KUKA KRL program: EPS_2_25694_WD01A_A_20260120031656.src

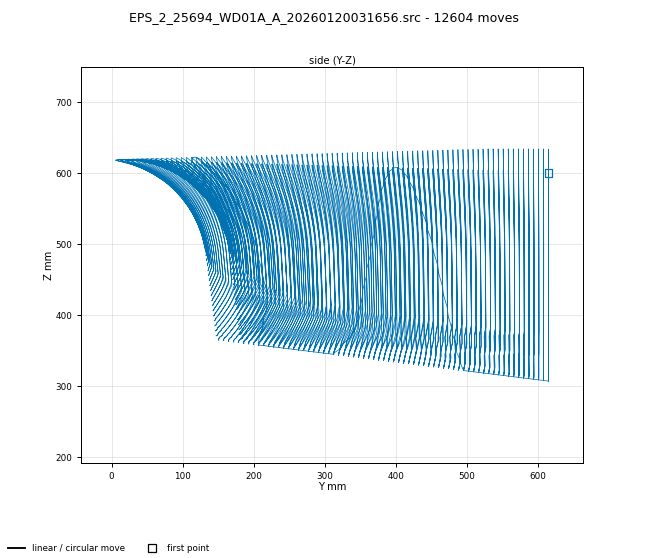
[picture p0: tool path of EPS_2_25694_WD01A_A_20260120031656.src, 12604 of 12606 moves have a stored position in this frame; points joined in program order, loops and branches not executed]
&ACCESS RVP
&REL 4
&COMMENT QRS 19112012
&PARAM EDITMASK = *
DEF PART()
EXT BAS (BAS_COMMAND :IN,REAL :IN )
INT I
BAS (#INITMOV,0 )

;KUKA QRS Post kuka4.cps  Date:22-06-2017 !

File_ID=2994

QRS_PRE_INIT()

;Init var - Until changes are made in qrs_pre_init
Outlet_Square_prg=0
Inlet_1_Square_prg=0
Inlet_2_Square_prg=0
Inlet_3_Square_prg=0
Inlet_4_Square_prg=0
Inlet_5_Square_prg=0

Outlet_1={X 0.000, Y 527.380, Z 509.000, B 0.000, E1 0.000 }
Inlet_1={X 0.000, Y 529.540, Z 479.000, B 0.000, E1 175.000 }
Outlet_1_type=251
Inlet_1_type=251
;QRS#1=Sidecore dimensions
;QRS#2=250-10" PVC SDR 35
;QRS#3=250-10" PVC SDR 35
;QRS#4=
;QRS#5=
;QRS#6=
;QRS#7=
;QRS#8=
;QRS#9=14M PSX
;QRS#10=14M PSX
;QRS#11=
;QRS#12=
;QRS#13=
;QRS#14=
;QRS#15=
;QRS#16=1220x127x914 3'
;QRS#17=EPS Height
;QRS#18=634,5
;QRS#19=*
;QRS#20= UPDATED VERSION 22-06-2017
;QRS#21=*
Outlet_Square=0100
Inlet_1_Square=0100
Inlet_2_Square=0
Inlet_3_Square=0
Inlet_4_Square=0
Inlet_5_Square=0
Mill_Square=1
Outlet_Square_Prg=205
Inlet_1_Square_prg=205

QRS_INIT()

$ADVANCE=5

; T1
PTP {E1 173.652,E2 173.652}
PTP {X 0,Y 615.445,A -85,B 0,C 180,E1 173.652,E2 173.652,E3 0,E4 0,E5 0,E6 0}
QRS_SPEED_INIT()
LIN {X 0,Y 615.445,Z 600,A -85,B 0,C 180,E1 173.652,E2 173.652,E3 0,E4 0,E5 0,E6 0} C_VEL
LIN {X 0,Y 615.445,Z 317.5,A -85,B 0,C 180,E1 173.652,E2 173.652} C_VEL
LIN {X 0,Y 615.445,Z 309.32,A -85,B 0,C 180,E1 173.652,E2 173.652} C_VEL
LIN {X 0,Y 615.438,Z 307.32,A -85,B 0,C 180,E1 173.466,E2 173.466} C_VEL
LIN {X 0,Y 615.464,Z 307.316,A -85,B 0,C 180,E1 170.801,E2 170.801} C_VEL
LIN {X 0,Y 615.478,Z 307.325,A -85,B 0,C 180,E1 168.139,E2 168.139} C_VEL
LIN {X 0,Y 615.433,Z 307.32,A -85,B 0,C 180,E1 165.449,E2 165.449} C_VEL
LIN {X 0,Y 615.481,Z 307.316,A -85,B 0,C 180,E1 162.729,E2 162.729} C_VEL
LIN {X 0,Y 615.451,Z 307.323,A -85,B 0,C 180,E1 159.966,E2 159.966} C_VEL
LIN {X 0,Y 615.43,Z 307.322,A -85,B 0,C 180,E1 157.668,E2 157.668} C_VEL
LIN {X 0,Y 615.429,Z 307.322,A -85,B 0,C 180,E1 155.725,E2 155.725} C_VEL
LIN {X 0,Y 615.426,Z 307.322,A -85,B 0,C 180,E1 153.553,E2 153.553} C_VEL
LIN {X 0,Y 615.493,Z 307.323,A -85,B 0,C 180,E1 150.594,E2 150.594} C_VEL
LIN {X 0,Y 615.471,Z 307.324,A -85,B 0,C 180,E1 148.313,E2 148.313} C_VEL
LIN {X 0,Y 615.433,Z 307.323,A -85,B 0,C 180,E1 145.974,E2 145.974} C_VEL
LIN {X 0,Y 615.421,Z 307.322,A -85,B 0,C 180,E1 143.57,E2 143.57} C_VEL
LIN {X 0,Y 615.463,Z 307.322,A -85,B 0,C 180,E1 140.941,E2 140.941} C_VEL
LIN {X 0,Y 615.482,Z 307.325,A -85,B 0,C 180,E1 138.525,E2 138.525} C_VEL
LIN {X 0,Y 615.424,Z 307.324,A -85,B 0,C 180,E1 136.009,E2 136.009} C_VEL
LIN {X 0,Y 615.421,Z 307.324,A -85,B 0,C 180,E1 133.99,E2 133.99} C_VEL
LIN {X 0,Y 615.419,Z 307.324,A -85,B 0,C 180,E1 131.48,E2 131.48} C_VEL
LIN {X 0,Y 615.473,Z 307.326,A -85,B 0,C 180,E1 128.906,E2 128.906} C_VEL
LIN {X 0,Y 615.446,Z 307.325,A -85,B 0,C 180,E1 126.428,E2 126.428} C_VEL
LIN {X 0,Y 615.414,Z 307.325,A -85,B 0,C 180,E1 124.027,E2 124.027} C_VEL
LIN {X 0,Y 615.412,Z 307.325,A -85,B 0,C 180,E1 121.69,E2 121.69} C_VEL
LIN {X 0,Y 615.428,Z 307.325,A -85,B 0,C 180,E1 119.41,E2 119.41} C_VEL
LIN {X 0,Y 615.444,Z 307.323,A -85,B 0,C 180,E1 116.446,E2 116.446} C_VEL
LIN {X 0,Y 615.423,Z 307.397,A -85,B 0,C 180,E1 115.597,E2 115.597} C_VEL
LIN {X 0,Y 615.49,Z 326.441,A -85,B 0,C 180,E1 112.845,E2 112.845} C_VEL
LIN {X 0,Y 615.48,Z 342.634,A -85,B 0,C 180,E1 110.538,E2 110.538} C_VEL
LIN {X 0,Y 615.496,Z 479.164,A -85,B 0,C 180,E1 108.905,E2 108.905} C_VEL
LIN {X 0,Y 615.495,Z 493.339,A -85,B 0,C 180,E1 108.605,E2 108.605} C_VEL
LIN {X 0,Y 615.494,Z 506.524,A -85,B 0,C 180,E1 108.2,E2 108.2} C_VEL
LIN {X 0,Y 615.497,Z 518.867,A -85,B 0,C 180,E1 107.699,E2 107.699} C_VEL
LIN {X 0,Y 615.492,Z 532.079,A -85,B 0,C 180,E1 107.014,E2 107.014} C_VEL
LIN {X 0,Y 615.498,Z 543.22,A -85,B 0,C 180,E1 106.301,E2 106.301} C_VEL
LIN {X 0,Y 615.499,Z 554.818,A -85,B 0,C 180,E1 105.395,E2 105.395} C_VEL
LIN {X 0,Y 615.496,Z 565.347,A -85,B 0,C 180,E1 104.395,E2 104.395} C_VEL
LIN {X 0,Y 615.497,Z 574.255,A -85,B 0,C 180,E1 103.369,E2 103.369} C_VEL
LIN {X 0,Y 615.496,Z 582.577,A -85,B 0,C 180,E1 102.195,E2 102.195} C_VEL
LIN {X 0,Y 615.496,Z 588.372,A -85,B 0,C 180,E1 101.193,E2 101.193} C_VEL
LIN {X 0,Y 615.497,Z 593.088,A -85,B 0,C 180,E1 100.194,E2 100.194} C_VEL
LIN {X 0,Y 615.497,Z 597.952,A -85,B 0,C 180,E1 98.868,E2 98.868} C_VEL
LIN {X 0,Y 615.496,Z 600.595,A -85,B 0,C 180,E1 97.876,E2 97.876} C_VEL
LIN {X 0,Y 615.495,Z 602.88,A -85,B 0,C 180,E1 96.557,E2 96.557} C_VEL
LIN {X 0,Y 615.489,Z 603.827,A -85,B 0,C 180,E1 95.241,E2 95.241} C_VEL
LIN {X 0,Y 615.493,Z 603.459,A -85,B 0,C 180,E1 93.929,E2 93.929} C_VEL
LIN {X 0,Y 615.491,Z 601.783,A -85,B 0,C 180,E1 92.618,E2 92.618} C_VEL
LIN {X 0,Y 615.495,Z 598.753,A -85,B 0,C 180,E1 91.309,E2 91.309} C_VEL
LIN {X 0,Y 615.496,Z 594.297,A -85,B 0,C 180,E1 90,E2 90} C_VEL
LIN {X 0,Y 615.495,Z 589.885,A -85,B 0,C 180,E1 89.019,E2 89.019} C_VEL
LIN {X 0,Y 615.499,Z 584.538,A -85,B 0,C 180,E1 88.037,E2 88.037} C_VEL
LIN {X 0,Y 615.496,Z 576.898,A -85,B 0,C 180,E1 86.891,E2 86.891} C_VEL
LIN {X 0,Y 615.496,Z 567.474,A -85,B 0,C 180,E1 85.744,E2 85.744} C_VEL
LIN {X 0,Y 615.498,Z 557.621,A -85,B 0,C 180,E1 84.759,E2 84.759} C_VEL
LIN {X 0,Y 615.499,Z 546.628,A -85,B 0,C 180,E1 83.855,E2 83.855} C_VEL
LIN {X 0,Y 615.491,Z 534.195,A -85,B 0,C 180,E1 83.022,E2 83.022} C_VEL
LIN {X 0,Y 615.494,Z 522.224,A -85,B 0,C 180,E1 82.372,E2 82.372} C_VEL
LIN {X 0,Y 615.493,Z 508.759,A -85,B 0,C 180,E1 81.794,E2 81.794} C_VEL
LIN {X 0,Y 615.495,Z 494.585,A -85,B 0,C 180,E1 81.339,E2 81.339} C_VEL
LIN {X 0,Y 615.495,Z 480.493,A -85,B 0,C 180,E1 81.029,E2 81.029} C_VEL
LIN {X 0,Y 615.476,Z 440.355,A -85,B 0,C 180,E1 80.532,E2 80.532} C_VEL
LIN {X 0,Y 615.486,Z 342.551,A -85,B 0,C 180,E1 79.361,E2 79.361} C_VEL
LIN {X 0,Y 615.487,Z 323.409,A -85,B 0,C 180,E1 76.631,E2 76.631} C_VEL
LIN {X 0,Y 615.424,Z 307.324,A -85,B 0,C 180,E1 74.284,E2 74.284} C_VEL
LIN {X 0,Y 615.414,Z 307.324,A -85,B 0,C 180,E1 72.041,E2 72.041} C_VEL
LIN {X 0,Y 615.476,Z 307.322,A -85,B 0,C 180,E1 69.269,E2 69.269} C_VEL
LIN {X 0,Y 615.424,Z 307.324,A -85,B 0,C 180,E1 66.441,E2 66.441} C_VEL
LIN {X 0,Y 615.414,Z 307.325,A -85,B 0,C 180,E1 64.281,E2 64.281} C_VEL
LIN {X 0,Y 615.409,Z 307.325,A -85,B 0,C 180,E1 62.081,E2 62.081} C_VEL
LIN {X 0,Y 615.485,Z 307.325,A -85,B 0,C 180,E1 59.08,E2 59.08} C_VEL
LIN {X 0,Y 615.416,Z 307.325,A -85,B 0,C 180,E1 56.477,E2 56.477} C_VEL
LIN {X 0,Y 615.413,Z 307.325,A -85,B 0,C 180,E1 54.379,E2 54.379} C_VEL
LIN {X 0,Y 615.422,Z 307.324,A -85,B 0,C 180,E1 51.926,E2 51.926} C_VEL
LIN {X 0,Y 615.469,Z 307.328,A -85,B 0,C 180,E1 49.392,E2 49.392} C_VEL
LIN {X 0,Y 615.436,Z 307.323,A -85,B 0,C 180,E1 46.751,E2 46.751} C_VEL
LIN {X 0,Y 615.418,Z 307.324,A -85,B 0,C 180,E1 44.156,E2 44.156} C_VEL
LIN {X 0,Y 615.425,Z 307.323,A -85,B 0,C 180,E1 42.073,E2 42.073} C_VEL
LIN {X 0,Y 615.453,Z 307.324,A -85,B 0,C 180,E1 39.753,E2 39.753} C_VEL
LIN {X 0,Y 615.451,Z 307.32,A -85,B 0,C 180,E1 36.932,E2 36.932} C_VEL
LIN {X 0,Y 615.432,Z 307.321,A -85,B 0,C 180,E1 34.693,E2 34.693} C_VEL
LIN {X 0,Y 615.426,Z 307.322,A -85,B 0,C 180,E1 32.321,E2 32.321} C_VEL
LIN {X 0,Y 615.464,Z 307.324,A -85,B 0,C 180,E1 29.79,E2 29.79} C_VEL
LIN {X 0,Y 615.459,Z 307.318,A -85,B 0,C 180,E1 27.039,E2 27.039} C_VEL
LIN {X 0,Y 615.449,Z 307.319,A -85,B 0,C 180,E1 24.994,E2 24.994} C_VEL
LIN {X 0,Y 615.437,Z 307.32,A -85,B 0,C 180,E1 22.847,E2 22.847} C_VEL
LIN {X 0,Y 615.431,Z 307.32,A -85,B 0,C 180,E1 20.542,E2 20.542} C_VEL
LIN {X 0,Y 615.464,Z 307.323,A -85,B 0,C 180,E1 17.958,E2 17.958} C_VEL
LIN {X 0,Y 615.474,Z 307.316,A -85,B 0,C 180,E1 15.227,E2 15.227} C_VEL
LIN {X 0,Y 615.436,Z 307.32,A -85,B 0,C 180,E1 12.531,E2 12.531} C_VEL
LIN {X 0,Y 615.489,Z 307.325,A -85,B 0,C 180,E1 9.862,E2 9.862} C_VEL
LIN {X 0,Y 615.469,Z 307.315,A -85,B 0,C 180,E1 7.216,E2 7.216} C_VEL
LIN {X 0,Y 615.44,Z 307.319,A -85,B 0,C 180,E1 4.585,E2 4.585} C_VEL
LIN {X 0,Y 615.489,Z 307.324,A -85,B 0,C 180,E1 1.963,E2 1.963} C_VEL
LIN {X 0,Y 615.477,Z 307.314,A -85,B 0,C 180,E1 -0.654,E2 -0.654} C_VEL
LIN {X 0,Y 615.441,Z 307.319,A -85,B 0,C 180,E1 -3.273,E2 -3.273} C_VEL
LIN {X 0,Y 615.483,Z 307.324,A -85,B 0,C 180,E1 -5.898,E2 -5.898} C_VEL
LIN {X 0,Y 615.482,Z 307.313,A -85,B 0,C 180,E1 -8.537,E2 -8.537} C_VEL
LIN {X 0,Y 615.447,Z 307.318,A -85,B 0,C 180,E1 -11.194,E2 -11.194} C_VEL
LIN {X 0,Y 615.498,Z 307.325,A -85,B 0,C 180,E1 -13.935,E2 -13.935} C_VEL
LIN {X 0,Y 615.476,Z 307.312,A -85,B 0,C 180,E1 -16.587,E2 -16.587} C_VEL
LIN {X 0,Y 615.472,Z 307.312,A -85,B 0,C 180,E1 -18.646,E2 -18.646} C_VEL
LIN {X 0,Y 615.465,Z 307.313,A -85,B 0,C 180,E1 -20.731,E2 -20.731} C_VEL
LIN {X 0,Y 615.458,Z 307.314,A -85,B 0,C 180,E1 -22.846,E2 -22.846} C_VEL
LIN {X 0,Y 615.477,Z 307.323,A -85,B 0,C 180,E1 -25.566,E2 -25.566} C_VEL
LIN {X 0,Y 615.488,Z 307.309,A -85,B 0,C 180,E1 -28.45,E2 -28.45} C_VEL
LIN {X 0,Y 615.457,Z 307.317,A -85,B 0,C 180,E1 -31.081,E2 -31.081} C_VEL
LIN {X 0,Y 615.479,Z 307.324,A -85,B 0,C 180,E1 -33.532,E2 -33.532} C_VEL
LIN {X 0,Y 615.484,Z 307.309,A -85,B 0,C 180,E1 -36.425,E2 -36.425} C_VEL
LIN {X 0,Y 615.461,Z 307.317,A -85,B 0,C 180,E1 -39.059,E2 -39.059} C_VEL
LIN {X 0,Y 615.486,Z 307.324,A -85,B 0,C 180,E1 -41.474,E2 -41.474} C_VEL
LIN {X 0,Y 615.494,Z 307.309,A -85,B 0,C 180,E1 -44.149,E2 -44.149} C_VEL
LIN {X 0,Y 615.463,Z 307.317,A -85,B 0,C 180,E1 -46.955,E2 -46.955} C_VEL
LIN {X 0,Y 615.491,Z 307.324,A -85,B 0,C 180,E1 -49.394,E2 -49.394} C_VEL
LIN {X 0,Y 615.488,Z 307.312,A -85,B 0,C 180,E1 -51.988,E2 -51.988} C_VEL
LIN {X 0,Y 615.483,Z 307.308,A -85,B 0,C 180,E1 -54.384,E2 -54.384} C_VEL
LIN {X 0,Y 615.467,Z 307.315,A -85,B 0,C 180,E1 -56.762,E2 -56.762} C_VEL
LIN {X 0,Y 615.476,Z 307.321,A -85,B 0,C 180,E1 -59.079,E2 -59.079} C_VEL
LIN {X 0,Y 615.487,Z 307.32,A -85,B 0,C 180,E1 -61.55,E2 -61.55} C_VEL
LIN {X 0,Y 615.477,Z 307.31,A -85,B 0,C 180,E1 -64.433,E2 -64.433} C_VEL
LIN {X 0,Y 615.474,Z 307.366,A -85,B 0,C 180,E1 -66.51,E2 -66.51} C_VEL
LIN {X 0,Y 615.496,Z 329.445,A -85,B 0,C 180,E1 -69.269,E2 -69.269} C_VEL
LIN {X 0,Y 615.498,Z 352.034,A -85,B 0,C 180,E1 -72.043,E2 -72.043} C_VEL
LIN {X 0,Y 615.49,Z 371.425,A -85,B 0,C 180,E1 -74.392,E2 -74.392} C_VEL
LIN {X 0,Y 615.498,Z 509.933,A -85,B 0,C 180,E1 -76.064,E2 -76.064} C_VEL
LIN {X 0,Y 615.495,Z 524.374,A -85,B 0,C 180,E1 -76.378,E2 -76.378} C_VEL
LIN {X 0,Y 615.489,Z 537.686,A -85,B 0,C 180,E1 -76.799,E2 -76.799} C_VEL
LIN {X 0,Y 615.498,Z 551.58,A -85,B 0,C 180,E1 -77.386,E2 -77.386} C_VEL
LIN {X 0,Y 615.495,Z 564.006,A -85,B 0,C 180,E1 -78.056,E2 -78.056} C_VEL
LIN {X 0,Y 615.499,Z 575.339,A -85,B 0,C 180,E1 -78.807,E2 -78.807} C_VEL
LIN {X 0,Y 615.498,Z 585.747,A -85,B 0,C 180,E1 -79.64,E2 -79.64} C_VEL
LIN {X 0,Y 615.496,Z 596.088,A -85,B 0,C 180,E1 -80.636,E2 -80.636} C_VEL
LIN {X 0,Y 615.497,Z 604.602,A -85,B 0,C 180,E1 -81.629,E2 -81.629} C_VEL
LIN {X 0,Y 615.496,Z 612.726,A -85,B 0,C 180,E1 -82.784,E2 -82.784} C_VEL
LIN {X 0,Y 615.496,Z 618.43,A -85,B 0,C 180,E1 -83.773,E2 -83.773} C_VEL
LIN {X 0,Y 615.495,Z 623.08,A -85,B 0,C 180,E1 -84.759,E2 -84.759} C_VEL
LIN {X 0,Y 615.494,Z 627.901,A -85,B 0,C 180,E1 -86.072,E2 -86.072} C_VEL
LIN {X 0,Y 615.496,Z 631.252,A -85,B 0,C 180,E1 -87.382,E2 -87.382} C_VEL
LIN {X 0,Y 615.489,Z 633.229,A -85,B 0,C 180,E1 -88.691,E2 -88.691} C_VEL
LIN {X 0,Y 615.493,Z 633.889,A -85,B 0,C 180,E1 -90,E2 -90} C_VEL
LIN {X 0,Y 615.489,Z 633.229,A -85,B 0,C 180,E1 -91.309,E2 -91.309} C_VEL
LIN {X 0,Y 615.496,Z 631.252,A -85,B 0,C 180,E1 -92.618,E2 -92.618} C_VEL
LIN {X 0,Y 615.494,Z 627.901,A -85,B 0,C 180,E1 -93.929,E2 -93.929} C_VEL
LIN {X 0,Y 615.495,Z 623.08,A -85,B 0,C 180,E1 -95.241,E2 -95.241} C_VEL
LIN {X 0,Y 615.496,Z 616.628,A -85,B 0,C 180,E1 -96.557,E2 -96.557} C_VEL
LIN {X 0,Y 615.497,Z 609.44,A -85,B 0,C 180,E1 -97.711,E2 -97.711} C_VEL
LIN {X 0,Y 615.497,Z 601.902,A -85,B 0,C 180,E1 -98.702,E2 -98.702} C_VEL
LIN {X 0,Y 615.495,Z 592.851,A -85,B 0,C 180,E1 -99.696,E2 -99.696} C_VEL
LIN {X 0,Y 615.497,Z 582.756,A -85,B 0,C 180,E1 -100.618,E2 -100.618} C_VEL
LIN {X 0,Y 615.498,Z 571.855,A -85,B 0,C 180,E1 -101.443,E2 -101.443} C_VEL
LIN {X 0,Y 615.489,Z 559.703,A -85,B 0,C 180,E1 -102.195,E2 -102.195} C_VEL
LIN {X 0,Y 615.498,Z 546.086,A -85,B 0,C 180,E1 -102.865,E2 -102.865} C_VEL
LIN {X 0,Y 615.49,Z 532.829,A -85,B 0,C 180,E1 -103.369,E2 -103.369} C_VEL
LIN {X 0,Y 615.494,Z 519.278,A -85,B 0,C 180,E1 -103.748,E2 -103.748} C_VEL
LIN {X 0,Y 615.494,Z 504.739,A -85,B 0,C 180,E1 -104.013,E2 -104.013} C_VEL
LIN {X 0,Y 615.49,Z 371.425,A -85,B 0,C 180,E1 -105.608,E2 -105.608} C_VEL
LIN {X 0,Y 615.485,Z 348.06,A -85,B 0,C 180,E1 -108.442,E2 -108.442} C_VEL
LIN {X 0,Y 615.489,Z 325.206,A -85,B 0,C 180,E1 -111.256,E2 -111.256} C_VEL
LIN {X 0,Y 615.475,Z 307.311,A -85,B 0,C 180,E1 -113.512,E2 -113.512} C_VEL
LIN {X 0,Y 615.487,Z 307.307,A -85,B 0,C 180,E1 -115.716,E2 -115.716} C_VEL
LIN {X 0,Y 615.486,Z 307.328,A -85,B 0,C 180,E1 -118.658,E2 -118.658} C_VEL
LIN {X 0,Y 615.469,Z 307.318,A -85,B 0,C 180,E1 -121.083,E2 -121.083} C_VEL
LIN {X 0,Y 615.476,Z 307.31,A -85,B 0,C 180,E1 -123.532,E2 -123.532} C_VEL
LIN {X 0,Y 615.483,Z 307.324,A -85,B 0,C 180,E1 -126.425,E2 -126.425} C_VEL
LIN {X 0,Y 615.465,Z 307.317,A -85,B 0,C 180,E1 -129.059,E2 -129.059} C_VEL
LIN {X 0,Y 615.474,Z 307.31,A -85,B 0,C 180,E1 -131.475,E2 -131.475} C_VEL
LIN {X 0,Y 615.487,Z 307.317,A -85,B 0,C 180,E1 -134.15,E2 -134.15} C_VEL
LIN {X 0,Y 615.463,Z 307.318,A -85,B 0,C 180,E1 -136.956,E2 -136.956} C_VEL
LIN {X 0,Y 615.47,Z 307.311,A -85,B 0,C 180,E1 -139.392,E2 -139.392} C_VEL
LIN {X 0,Y 615.49,Z 307.315,A -85,B 0,C 180,E1 -141.988,E2 -141.988} C_VEL
LIN {X 0,Y 615.495,Z 307.325,A -85,B 0,C 180,E1 -144.385,E2 -144.385} C_VEL
LIN {X 0,Y 615.459,Z 307.32,A -85,B 0,C 180,E1 -146.762,E2 -146.762} C_VEL
LIN {X 0,Y 615.457,Z 307.315,A -85,B 0,C 180,E1 -149.079,E2 -149.079} C_VEL
LIN {X 0,Y 615.488,Z 307.309,A -85,B 0,C 180,E1 -151.551,E2 -151.551} C_VEL
LIN {X 0,Y 615.476,Z 307.323,A -85,B 0,C 180,E1 -154.435,E2 -154.435} C_VEL
LIN {X 0,Y 615.458,Z 307.314,A -85,B 0,C 180,E1 -157.154,E2 -157.154} C_VEL
LIN {X 0,Y 615.493,Z 307.32,A -85,B 0,C 180,E1 -159.968,E2 -159.968} C_VEL
LIN {X 0,Y 615.451,Z 307.319,A -85,B 0,C 180,E1 -162.729,E2 -162.729} C_VEL
LIN {X 0,Y 615.484,Z 307.311,A -85,B 0,C 180,E1 -165.451,E2 -165.451} C_VEL
LIN {X 0,Y 615.484,Z 307.325,A -85,B 0,C 180,E1 -168.139,E2 -168.139} C_VEL
LIN {X 0,Y 615.446,Z 307.318,A -85,B 0,C 180,E1 -170.801,E2 -170.801} C_VEL
LIN {X 0,Y 615.488,Z 307.312,A -85,B 0,C 180,E1 -173.443,E2 -173.443} C_VEL
LIN {X 0,Y 615.48,Z 307.325,A -85,B 0,C 180,E1 -176.072,E2 -176.072} C_VEL
LIN {X 0,Y 615.441,Z 307.319,A -85,B 0,C 180,E1 -178.691,E2 -178.691} C_VEL
LIN {X 0,Y 615.476,Z 307.314,A -85,B 0,C 180,E1 -181.309,E2 -181.309} C_VEL
LIN {X 0,Y 615.481,Z 307.326,A -85,B 0,C 180,E1 -183.929,E2 -183.929} C_VEL
LIN {X 0,Y 615.438,Z 307.32,A -85,B 0,C 180,E1 -186.534,E2 -186.534} C_VEL
LIN {X 0,Y 614.78,Z 307.464,A -85,B 0,C 180,E1 -187.08,E2 -187.08} C_VEL
LIN {X 0,Y 611.959,Z 307.883,A -85,B 0,C 180,E1 -187.966,E2 -187.966} C_VEL
LIN {X 0,Y 609.57,Z 308.19,A -85,B 0,C 180,E1 -188.679,E2 -188.679} C_VEL
LIN {X 0,Y 608.536,Z 308.306,A -85,B 0,C 180,E1 -189.229,E2 -189.229} C_VEL
LIN {X 0,Y 608.447,Z 308.316,A -85,B 0,C 180,E1 -189.415,E2 -189.415} C_VEL
LIN {X 0,Y 608.447,Z 308.319,A -85,B 0,C 180,E1 -192,E2 -192} C_VEL
LIN {X 0,Y 608.407,Z 308.318,A -85,B 0,C 180,E1 -194.722,E2 -194.722} C_VEL
LIN {X 0,Y 608.443,Z 308.321,A -85,B 0,C 180,E1 -197.477,E2 -197.477} C_VEL
LIN {X 0,Y 608.42,Z 308.318,A -85,B 0,C 180,E1 -200.276,E2 -200.276} C_VEL
LIN {X 0,Y 608.399,Z 308.319,A -85,B 0,C 180,E1 -202.461,E2 -202.461} C_VEL
LIN {X 0,Y 608.413,Z 308.317,A -85,B 0,C 180,E1 -204.573,E2 -204.573} C_VEL
LIN {X 0,Y 608.464,Z 308.316,A -85,B 0,C 180,E1 -207.204,E2 -207.204} C_VEL
LIN {X 0,Y 608.419,Z 308.319,A -85,B 0,C 180,E1 -209.963,E2 -209.963} C_VEL
LIN {X 0,Y 608.408,Z 308.318,A -85,B 0,C 180,E1 -212.514,E2 -212.514} C_VEL
LIN {X 0,Y 608.409,Z 308.32,A -85,B 0,C 180,E1 -214.899,E2 -214.899} C_VEL
LIN {X 0,Y 608.435,Z 308.319,A -85,B 0,C 180,E1 -217.749,E2 -217.749} C_VEL
LIN {X 0,Y 608.406,Z 308.318,A -85,B 0,C 180,E1 -220.323,E2 -220.323} C_VEL
LIN {X 0,Y 608.428,Z 308.32,A -85,B 0,C 180,E1 -222.963,E2 -222.963} C_VEL
LIN {X 0,Y 608.411,Z 308.321,A -85,B 0,C 180,E1 -225.741,E2 -225.741} C_VEL
LIN {X 0,Y 608.409,Z 308.319,A -85,B 0,C 180,E1 -227.934,E2 -227.934} C_VEL
LIN {X 0,Y 608.414,Z 308.32,A -85,B 0,C 180,E1 -230.71,E2 -230.71} C_VEL
LIN {X 0,Y 608.433,Z 308.323,A -85,B 0,C 180,E1 -233.083,E2 -233.083} C_VEL
LIN {X 0,Y 608.447,Z 308.318,A -85,B 0,C 180,E1 -235.529,E2 -235.529} C_VEL
LIN {X 0,Y 608.412,Z 308.318,A -85,B 0,C 180,E1 -237.902,E2 -237.902} C_VEL
LIN {X 0,Y 608.401,Z 308.319,A -85,B 0,C 180,E1 -240.217,E2 -240.217} C_VEL
LIN {X 0,Y 608.441,Z 308.32,A -85,B 0,C 180,E1 -242.801,E2 -242.801} C_VEL
LIN {X 0,Y 608.399,Z 308.36,A -85,B 0,C 180,E1 -244.294,E2 -244.294} C_VEL
LIN {X 0,Y 608.505,Z 322.308,A -85,B 0,C 180,E1 -246.337,E2 -246.337} C_VEL
LIN {X 0,Y 608.508,Z 340.913,A -85,B 0,C 180,E1 -249.02,E2 -249.02} C_VEL
LIN {X 0,Y 608.508,Z 342.73,A -85,B 0,C 180,E1 -249.28,E2 -249.28} C_VEL
LIN {X 0,Y 608.613,Z 479.428,A -85,B 0,C 180,E1 -250.939,E2 -250.939} C_VEL
LIN {X 0,Y 608.589,Z 493.905,A -85,B 0,C 180,E1 -251.253,E2 -251.253} C_VEL
LIN {X 0,Y 608.561,Z 508.178,A -85,B 0,C 180,E1 -251.709,E2 -251.709} C_VEL
LIN {X 0,Y 608.543,Z 521.237,A -85,B 0,C 180,E1 -252.266,E2 -252.266} C_VEL
LIN {X 0,Y 608.531,Z 534.035,A -85,B 0,C 180,E1 -252.959,E2 -252.959} C_VEL
LIN {X 0,Y 608.51,Z 546.187,A -85,B 0,C 180,E1 -253.774,E2 -253.774} C_VEL
LIN {X 0,Y 608.491,Z 556.282,A -85,B 0,C 180,E1 -254.594,E2 -254.594} C_VEL
LIN {X 0,Y 608.475,Z 566.799,A -85,B 0,C 180,E1 -255.621,E2 -255.621} C_VEL
LIN {X 0,Y 608.462,Z 575.427,A -85,B 0,C 180,E1 -256.643,E2 -256.643} C_VEL
LIN {X 0,Y 608.44,Z 583.63,A -85,B 0,C 180,E1 -257.83,E2 -257.83} C_VEL
LIN {X 0,Y 608.432,Z 590.464,A -85,B 0,C 180,E1 -259.065,E2 -259.065} C_VEL
LIN {X 0,Y 608.43,Z 596.015,A -85,B 0,C 180,E1 -260.358,E2 -260.358} C_VEL
LIN {X 0,Y 608.426,Z 599.325,A -85,B 0,C 180,E1 -261.363,E2 -261.363} C_VEL
LIN {X 0,Y 608.421,Z 602.402,A -85,B 0,C 180,E1 -262.7,E2 -262.7} C_VEL
LIN {X 0,Y 608.433,Z 604.085,A -85,B 0,C 180,E1 -264.033,E2 -264.033} C_VEL
LIN {X 0,Y 608.423,Z 604.432,A -85,B 0,C 180,E1 -265.362,E2 -265.362} C_VEL
LIN {X 0,Y 608.416,Z 603.453,A -85,B 0,C 180,E1 -266.689,E2 -266.689} C_VEL
LIN {X 0,Y 608.444,Z 601.137,A -85,B 0,C 180,E1 -268.014,E2 -268.014} C_VEL
LIN {X 0,Y 608.437,Z 597.424,A -85,B 0,C 180,E1 -269.338,E2 -269.338} C_VEL
LIN {X 0,Y 608.437,Z 592.217,A -85,B 0,C 180,E1 -270.662,E2 -270.662} C_VEL
LIN {X 0,Y 608.441,Z 587.177,A -85,B 0,C 180,E1 -271.655,E2 -271.655} C_VEL
LIN {X 0,Y 608.446,Z 580.009,A -85,B 0,C 180,E1 -272.814,E2 -272.814} C_VEL
LIN {X 0,Y 608.455,Z 571.177,A -85,B 0,C 180,E1 -273.974,E2 -273.974} C_VEL
LIN {X 0,Y 608.474,Z 561.943,A -85,B 0,C 180,E1 -274.97,E2 -274.97} C_VEL
LIN {X 0,Y 608.498,Z 550.694,A -85,B 0,C 180,E1 -275.967,E2 -275.967} C_VEL
LIN {X 0,Y 608.536,Z 538.524,A -85,B 0,C 180,E1 -276.849,E2 -276.849} C_VEL
LIN {X 0,Y 608.542,Z 526.683,A -85,B 0,C 180,E1 -277.549,E2 -277.549} C_VEL
LIN {X 0,Y 608.575,Z 514.418,A -85,B 0,C 180,E1 -278.133,E2 -278.133} C_VEL
LIN {X 0,Y 608.598,Z 500.854,A -85,B 0,C 180,E1 -278.634,E2 -278.634} C_VEL
LIN {X 0,Y 608.601,Z 486.751,A -85,B 0,C 180,E1 -279.011,E2 -279.011} C_VEL
LIN {X 0,Y 608.599,Z 473.246,A -85,B 0,C 180,E1 -279.241,E2 -279.241} C_VEL
LIN {X 0,Y 608.495,Z 342.746,A -85,B 0,C 180,E1 -280.808,E2 -280.808} C_VEL
LIN {X 0,Y 608.527,Z 323.87,A -85,B 0,C 180,E1 -283.525,E2 -283.525} C_VEL
LIN {X 0,Y 608.409,Z 308.367,A -85,B 0,C 180,E1 -285.794,E2 -285.794} C_VEL
LIN {X 0,Y 608.435,Z 308.321,A -85,B 0,C 180,E1 -288.705,E2 -288.705} C_VEL
LIN {X 0,Y 608.438,Z 308.325,A -85,B 0,C 180,E1 -290.982,E2 -290.982} C_VEL
LIN {X 0,Y 608.423,Z 308.323,A -85,B 0,C 180,E1 -293.125,E2 -293.125} C_VEL
LIN {X 0,Y 608.396,Z 308.32,A -85,B 0,C 180,E1 -295.705,E2 -295.705} C_VEL
LIN {X 0,Y 608.395,Z 308.321,A -85,B 0,C 180,E1 -298.27,E2 -298.27} C_VEL
LIN {X 0,Y 608.435,Z 308.318,A -85,B 0,C 180,E1 -301.265,E2 -301.265} C_VEL
LIN {X 0,Y 608.379,Z 308.321,A -85,B 0,C 180,E1 -303.721,E2 -303.721} C_VEL
LIN {X 0,Y 608.392,Z 308.321,A -85,B 0,C 180,E1 -306.096,E2 -306.096} C_VEL
LIN {X 0,Y 608.411,Z 308.326,A -85,B 0,C 180,E1 -308.593,E2 -308.593} C_VEL
LIN {X 0,Y 608.416,Z 308.318,A -85,B 0,C 180,E1 -311.337,E2 -311.337} C_VEL
LIN {X 0,Y 608.417,Z 308.317,A -85,B 0,C 180,E1 -313.875,E2 -313.875} C_VEL
LIN {X 0,Y 608.481,Z 308.319,A -85,B 0,C 180,E1 -316.691,E2 -316.691} C_VEL
LIN {X 0,Y 608.443,Z 308.32,A -85,B 0,C 180,E1 -318.822,E2 -318.822} C_VEL
LIN {X 0,Y 608.398,Z 308.319,A -85,B 0,C 180,E1 -321.406,E2 -321.406} C_VEL
LIN {X 0,Y 608.432,Z 308.317,A -85,B 0,C 180,E1 -323.957,E2 -323.957} C_VEL
LIN {X 0,Y 608.448,Z 308.32,A -85,B 0,C 180,E1 -326.328,E2 -326.328} C_VEL
LIN {X 0,Y 608.443,Z 308.32,A -85,B 0,C 180,E1 -328.734,E2 -328.734} C_VEL
LIN {X 0,Y 608.426,Z 308.316,A -85,B 0,C 180,E1 -331.389,E2 -331.389} C_VEL
LIN {X 0,Y 608.418,Z 308.32,A -85,B 0,C 180,E1 -333.963,E2 -333.963} C_VEL
LIN {X 0,Y 608.427,Z 308.318,A -85,B 0,C 180,E1 -336.875,E2 -336.875} C_VEL
LIN {X 0,Y 608.427,Z 308.315,A -85,B 0,C 180,E1 -339.333,E2 -339.333} C_VEL
LIN {X 0,Y 608.416,Z 308.319,A -85,B 0,C 180,E1 -341.827,E2 -341.827} C_VEL
LIN {X 0,Y 608.46,Z 308.317,A -85,B 0,C 180,E1 -344.594,E2 -344.594} C_VEL
LIN {X 0,Y 608.412,Z 308.317,A -85,B 0,C 180,E1 -347.321,E2 -347.321} C_VEL
LIN {X 0,Y 608.45,Z 308.319,A -85,B 0,C 180,E1 -350.022,E2 -350.022} C_VEL
LIN {X 0,Y 608.439,Z 308.317,A -85,B 0,C 180,E1 -352.7,E2 -352.7} C_VEL
LIN {X 0,Y 608.412,Z 308.318,A -85,B 0,C 180,E1 -355.362,E2 -355.362} C_VEL
LIN {X 0,Y 608.457,Z 308.321,A -85,B 0,C 180,E1 -358.014,E2 -358.014} C_VEL
LIN {X 0,Y 608.472,Z 308.312,A -85,B 0,C 180,E1 -360.662,E2 -360.662} C_VEL
LIN {X 0,Y 608.412,Z 308.318,A -85,B 0,C 180,E1 -363.311,E2 -363.311} C_VEL
LIN {X 0,Y 608.458,Z 308.322,A -85,B 0,C 180,E1 -365.967,E2 -365.967} C_VEL
LIN {X 0,Y 608.448,Z 308.314,A -85,B 0,C 180,E1 -368.636,E2 -368.636} C_VEL
LIN {X 0,Y 608.426,Z 308.317,A -85,B 0,C 180,E1 -371.325,E2 -371.325} C_VEL
LIN {X 0,Y 608.475,Z 308.318,A -85,B 0,C 180,E1 -374.037,E2 -374.037} C_VEL
LIN {X 0,Y 608.434,Z 308.315,A -85,B 0,C 180,E1 -376.784,E2 -376.784} C_VEL
LIN {X 0,Y 608.437,Z 308.32,A -85,B 0,C 180,E1 -379.571,E2 -379.571} C_VEL
LIN {X 0,Y 608.463,Z 308.312,A -85,B 0,C 180,E1 -382.476,E2 -382.476} C_VEL
LIN {X 0,Y 608.446,Z 308.314,A -85,B 0,C 180,E1 -384.571,E2 -384.571} C_VEL
LIN {X 0,Y 608.435,Z 308.317,A -85,B 0,C 180,E1 -387.198,E2 -387.198} C_VEL
LIN {X 0,Y 608.475,Z 308.316,A -85,B 0,C 180,E1 -389.972,E2 -389.972} C_VEL
LIN {X 0,Y 608.446,Z 308.314,A -85,B 0,C 180,E1 -392.88,E2 -392.88} C_VEL
LIN {X 0,Y 608.44,Z 308.318,A -85,B 0,C 180,E1 -395.278,E2 -395.278} C_VEL
LIN {X 0,Y 608.468,Z 308.312,A -85,B 0,C 180,E1 -398.24,E2 -398.24} C_VEL
LIN {X 0,Y 608.453,Z 308.319,A -85,B 0,C 180,E1 -401.341,E2 -401.341} C_VEL
LIN {X 0,Y 608.46,Z 308.312,A -85,B 0,C 180,E1 -404.264,E2 -404.264} C_VEL
LIN {X 0,Y 608.433,Z 308.318,A -85,B 0,C 180,E1 -407.038,E2 -407.038} C_VEL
LIN {X 0,Y 608.455,Z 308.319,A -85,B 0,C 180,E1 -409.697,E2 -409.697} C_VEL
LIN {X 0,Y 608.465,Z 308.311,A -85,B 0,C 180,E1 -412.253,E2 -412.253} C_VEL
LIN {X 0,Y 608.439,Z 308.315,A -85,B 0,C 180,E1 -414.722,E2 -414.722} C_VEL
LIN {X 0,Y 608.464,Z 308.32,A -85,B 0,C 180,E1 -417.477,E2 -417.477} C_VEL
LIN {X 0,Y 608.48,Z 308.309,A -85,B 0,C 180,E1 -420.221,E2 -420.221} C_VEL
LIN {X 0,Y 608.468,Z 308.313,A -85,B 0,C 180,E1 -422.795,E2 -422.795} C_VEL
LIN {X 0,Y 608.449,Z 308.322,A -85,B 0,C 180,E1 -425.429,E2 -425.429} C_VEL
LIN {X 0,Y 608.48,Z 308.426,A -85,B 0,C 180,E1 -426.359,E2 -426.359} C_VEL
LIN {X 0,Y 608.596,Z 325.206,A -85,B 0,C 180,E1 -428.491,E2 -428.491} C_VEL
LIN {X 0,Y 608.535,Z 347.483,A -85,B 0,C 180,E1 -431.267,E2 -431.267} C_VEL
LIN {X 0,Y 608.516,Z 371.131,A -85,B 0,C 180,E1 -434.166,E2 -434.166} C_VEL
LIN {X 0,Y 608.574,Z 372.029,A -85,B 0,C 180,E1 -434.232,E2 -434.232} C_VEL
LIN {X 0,Y 608.616,Z 509.892,A -85,B 0,C 180,E1 -435.902,E2 -435.902} C_VEL
LIN {X 0,Y 608.598,Z 524.381,A -85,B 0,C 180,E1 -436.221,E2 -436.221} C_VEL
LIN {X 0,Y 608.579,Z 537.708,A -85,B 0,C 180,E1 -436.646,E2 -436.646} C_VEL
LIN {X 0,Y 608.565,Z 549.881,A -85,B 0,C 180,E1 -437.155,E2 -437.155} C_VEL
LIN {X 0,Y 608.516,Z 562.679,A -85,B 0,C 180,E1 -437.832,E2 -437.832} C_VEL
LIN {X 0,Y 608.499,Z 575.469,A -85,B 0,C 180,E1 -438.677,E2 -438.677} C_VEL
LIN {X 0,Y 608.496,Z 585.93,A -85,B 0,C 180,E1 -439.519,E2 -439.519} C_VEL
LIN {X 0,Y 608.479,Z 596.334,A -85,B 0,C 180,E1 -440.527,E2 -440.527} C_VEL
LIN {X 0,Y 608.464,Z 604.913,A -85,B 0,C 180,E1 -441.531,E2 -441.531} C_VEL
LIN {X 0,Y 608.461,Z 613.113,A -85,B 0,C 180,E1 -442.701,E2 -442.701} C_VEL
LIN {X 0,Y 608.443,Z 619.545,A -85,B 0,C 180,E1 -443.831,E2 -443.831} C_VEL
LIN {X 0,Y 608.438,Z 624.962,A -85,B 0,C 180,E1 -445.03,E2 -445.03} C_VEL
LIN {X 0,Y 608.431,Z 628.441,A -85,B 0,C 180,E1 -446.026,E2 -446.026} C_VEL
LIN {X 0,Y 608.424,Z 631.831,A -85,B 0,C 180,E1 -447.352,E2 -447.352} C_VEL
LIN {X 0,Y 608.442,Z 633.83,A -85,B 0,C 180,E1 -448.676,E2 -448.676} C_VEL
LIN {X 0,Y 608.433,Z 634.5,A -85,B 0,C 180,E1 -450,E2 -450} C_VEL
LIN {X 0,Y 608.442,Z 633.83,A -85,B 0,C 180,E1 -451.324,E2 -451.324} C_VEL
LIN {X 0,Y 608.424,Z 631.831,A -85,B 0,C 180,E1 -452.648,E2 -452.648} C_VEL
LIN {X 0,Y 608.431,Z 628.441,A -85,B 0,C 180,E1 -453.974,E2 -453.974} C_VEL
LIN {X 0,Y 608.44,Z 623.567,A -85,B 0,C 180,E1 -455.302,E2 -455.302} C_VEL
LIN {X 0,Y 608.445,Z 617.211,A -85,B 0,C 180,E1 -456.604,E2 -456.604} C_VEL
LIN {X 0,Y 608.453,Z 609.797,A -85,B 0,C 180,E1 -457.8,E2 -457.8} C_VEL
LIN {X 0,Y 608.473,Z 600.822,A -85,B 0,C 180,E1 -458.971,E2 -458.971} C_VEL
LIN {X 0,Y 608.472,Z 591.389,A -85,B 0,C 180,E1 -459.977,E2 -459.977} C_VEL
LIN {X 0,Y 608.506,Z 580.047,A -85,B 0,C 180,E1 -460.973,E2 -460.973} C_VEL
LIN {X 0,Y 608.533,Z 568.145,A -85,B 0,C 180,E1 -461.829,E2 -461.829} C_VEL
LIN {X 0,Y 608.531,Z 555.069,A -85,B 0,C 180,E1 -462.591,E2 -462.591} C_VEL
LIN {X 0,Y 608.556,Z 542.168,A -85,B 0,C 180,E1 -463.185,E2 -463.185} C_VEL
LIN {X 0,Y 608.593,Z 528.174,A -85,B 0,C 180,E1 -463.673,E2 -463.673} C_VEL
LIN {X 0,Y 608.622,Z 514.442,A -85,B 0,C 180,E1 -464.013,E2 -464.013} C_VEL
LIN {X 0,Y 608.622,Z 498.148,A -85,B 0,C 180,E1 -464.258,E2 -464.258} C_VEL
LIN {X 0,Y 608.53,Z 371.572,A -85,B 0,C 180,E1 -465.78,E2 -465.78} C_VEL
LIN {X 0,Y 608.568,Z 346.402,A -85,B 0,C 180,E1 -468.866,E2 -468.866} C_VEL
LIN {X 0,Y 608.597,Z 323.792,A -85,B 0,C 180,E1 -471.687,E2 -471.687} C_VEL
LIN {X 0,Y 608.474,Z 308.337,A -85,B 0,C 180,E1 -473.653,E2 -473.653} C_VEL
LIN {X 0,Y 608.445,Z 308.315,A -85,B 0,C 180,E1 -476.036,E2 -476.036} C_VEL
LIN {X 0,Y 608.474,Z 308.32,A -85,B 0,C 180,E1 -478.62,E2 -478.62} C_VEL
LIN {X 0,Y 608.444,Z 308.314,A -85,B 0,C 180,E1 -481.318,E2 -481.318} C_VEL
LIN {X 0,Y 608.475,Z 308.31,A -85,B 0,C 180,E1 -483.735,E2 -483.735} C_VEL
LIN {X 0,Y 608.462,Z 308.314,A -85,B 0,C 180,E1 -486.091,E2 -486.091} C_VEL
LIN {X 0,Y 608.461,Z 308.321,A -85,B 0,C 180,E1 -488.589,E2 -488.589} C_VEL
LIN {X 0,Y 608.447,Z 308.313,A -85,B 0,C 180,E1 -491.341,E2 -491.341} C_VEL
LIN {X 0,Y 608.455,Z 308.319,A -85,B 0,C 180,E1 -494.264,E2 -494.264} C_VEL
LIN {X 0,Y 608.433,Z 308.316,A -85,B 0,C 180,E1 -497.038,E2 -497.038} C_VEL
LIN {X 0,Y 608.456,Z 308.313,A -85,B 0,C 180,E1 -499.697,E2 -499.697} C_VEL
LIN {X 0,Y 608.466,Z 308.319,A -85,B 0,C 180,E1 -502.254,E2 -502.254} C_VEL
LIN {X 0,Y 608.43,Z 308.316,A -85,B 0,C 180,E1 -505.098,E2 -505.098} C_VEL
LIN {X 0,Y 608.46,Z 308.312,A -85,B 0,C 180,E1 -507.479,E2 -507.479} C_VEL
LIN {X 0,Y 608.479,Z 308.319,A -85,B 0,C 180,E1 -510.221,E2 -510.221} C_VEL
LIN {X 0,Y 608.434,Z 308.317,A -85,B 0,C 180,E1 -512.802,E2 -512.802} C_VEL
LIN {X 0,Y 608.446,Z 308.314,A -85,B 0,C 180,E1 -515.429,E2 -515.429} C_VEL
LIN {X 0,Y 608.457,Z 308.32,A -85,B 0,C 180,E1 -518.308,E2 -518.308} C_VEL
LIN {X 0,Y 608.446,Z 308.313,A -85,B 0,C 180,E1 -521.13,E2 -521.13} C_VEL
LIN {X 0,Y 608.462,Z 308.318,A -85,B 0,C 180,E1 -523.906,E2 -523.906} C_VEL
LIN {X 0,Y 608.437,Z 308.316,A -85,B 0,C 180,E1 -526.643,E2 -526.643} C_VEL
LIN {X 0,Y 608.456,Z 308.313,A -85,B 0,C 180,E1 -529.35,E2 -529.35} C_VEL
LIN {X 0,Y 608.475,Z 308.32,A -85,B 0,C 180,E1 -532.033,E2 -532.033} C_VEL
LIN {X 0,Y 608.429,Z 308.316,A -85,B 0,C 180,E1 -534.698,E2 -534.698} C_VEL
LIN {X 0,Y 608.472,Z 308.312,A -85,B 0,C 180,E1 -537.352,E2 -537.352} C_VEL
LIN {X 0,Y 608.473,Z 308.319,A -85,B 0,C 180,E1 -540,E2 -540} C_VEL
LIN {X 0,Y 608.437,Z 308.315,A -85,B 0,C 180,E1 -542.648,E2 -542.648} C_VEL
LIN {X 0,Y 608.453,Z 308.315,A -85,B 0,C 180,E1 -545.302,E2 -545.302} C_VEL
LIN {X 0,Y 608.441,Z 308.321,A -85,B 0,C 180,E1 -547.968,E2 -547.968} C_VEL
LIN {X 0,Y 608.447,Z 308.316,A -85,B 0,C 180,E1 -549.415,E2 -549.415} C_VEL
LIN {X 0,Y 607.772,Z 308.405,A -85,B 0,C 180,E1 -549.967,E2 -549.967} C_VEL
LIN {X 0,Y 604.926,Z 308.758,A -85,B 0,C 180,E1 -550.864,E2 -550.864} C_VEL
LIN {X 0,Y 602.519,Z 309.059,A -85,B 0,C 180,E1 -551.585,E2 -551.585} C_VEL
LIN {X 0,Y 601.472,Z 309.186,A -85,B 0,C 180,E1 -552.142,E2 -552.142} C_VEL
LIN {X 0,Y 601.38,Z 309.195,A -85,B 0,C 180,E1 -552.33,E2 -552.33} C_VEL
LIN {X 0,Y 601.385,Z 309.193,A -85,B 0,C 180,E1 -554.898,E2 -554.898} C_VEL
LIN {X 0,Y 601.381,Z 309.204,A -85,B 0,C 180,E1 -557.689,E2 -557.689} C_VEL
LIN {X 0,Y 601.386,Z 309.2,A -85,B 0,C 180,E1 -559.81,E2 -559.81} C_VEL
LIN {X 0,Y 601.381,Z 309.198,A -85,B 0,C 180,E1 -561.961,E2 -561.961} C_VEL
LIN {X 0,Y 601.379,Z 309.194,A -85,B 0,C 180,E1 -564.88,E2 -564.88} C_VEL
LIN {X 0,Y 601.4,Z 309.198,A -85,B 0,C 180,E1 -567.359,E2 -567.359} C_VEL
LIN {X 0,Y 601.376,Z 309.194,A -85,B 0,C 180,E1 -570.167,E2 -570.167} C_VEL
LIN {X 0,Y 601.385,Z 309.193,A -85,B 0,C 180,E1 -572.709,E2 -572.709} C_VEL
LIN {X 0,Y 601.367,Z 309.2,A -85,B 0,C 180,E1 -575.107,E2 -575.107} C_VEL
LIN {X 0,Y 601.401,Z 309.201,A -85,B 0,C 180,E1 -577.422,E2 -577.422} C_VEL
LIN {X 0,Y 601.359,Z 309.198,A -85,B 0,C 180,E1 -580,E2 -580} C_VEL
LIN {X 0,Y 601.351,Z 309.198,A -85,B 0,C 180,E1 -582.584,E2 -582.584} C_VEL
LIN {X 0,Y 601.369,Z 309.195,A -85,B 0,C 180,E1 -584.529,E2 -584.529} C_VEL
LIN {X 0,Y 601.366,Z 309.204,A -85,B 0,C 180,E1 -587.415,E2 -587.415} C_VEL
LIN {X 0,Y 601.38,Z 309.194,A -85,B 0,C 180,E1 -590.472,E2 -590.472} C_VEL
LIN {X 0,Y 601.374,Z 309.201,A -85,B 0,C 180,E1 -593.415,E2 -593.415} C_VEL
LIN {X 0,Y 601.373,Z 309.195,A -85,B 0,C 180,E1 -596.074,E2 -596.074} C_VEL
LIN {X 0,Y 601.386,Z 309.195,A -85,B 0,C 180,E1 -598.552,E2 -598.552} C_VEL
LIN {X 0,Y 601.406,Z 309.197,A -85,B 0,C 180,E1 -601.372,E2 -601.372} C_VEL
LIN {X 0,Y 601.389,Z 309.27,A -85,B 0,C 180,E1 -604.177,E2 -604.177} C_VEL
LIN {X 0,Y 601.533,Z 317.851,A -85,B 0,C 180,E1 -605.455,E2 -605.455} C_VEL
LIN {X 0,Y 601.516,Z 335.515,A -85,B 0,C 180,E1 -608.045,E2 -608.045} C_VEL
LIN {X 0,Y 601.502,Z 342.731,A -85,B 0,C 180,E1 -609.092,E2 -609.092} C_VEL
LIN {X 0,Y 601.829,Z 348.492,A -85,B 0,C 180,E1 -609.174,E2 -609.174} C_VEL
LIN {X 0,Y 601.737,Z 479.679,A -85,B 0,C 180,E1 -610.779,E2 -610.779} C_VEL
LIN {X 0,Y 601.708,Z 493.942,A -85,B 0,C 180,E1 -611.093,E2 -611.093} C_VEL
LIN {X 0,Y 601.653,Z 506.853,A -85,B 0,C 180,E1 -611.502,E2 -611.502} C_VEL
LIN {X 0,Y 601.601,Z 519.987,A -85,B 0,C 180,E1 -612.054,E2 -612.054} C_VEL
LIN {X 0,Y 601.553,Z 533.024,A -85,B 0,C 180,E1 -612.755,E2 -612.755} C_VEL
LIN {X 0,Y 601.5,Z 545.504,A -85,B 0,C 180,E1 -613.591,E2 -613.591} C_VEL
LIN {X 0,Y 601.485,Z 555.59,A -85,B 0,C 180,E1 -614.41,E2 -614.41} C_VEL
LIN {X 0,Y 601.443,Z 566.235,A -85,B 0,C 180,E1 -615.449,E2 -615.449} C_VEL
LIN {X 0,Y 601.4,Z 574.972,A -85,B 0,C 180,E1 -616.484,E2 -616.484} C_VEL
LIN {X 0,Y 601.379,Z 583.271,A -85,B 0,C 180,E1 -617.685,E2 -617.685} C_VEL
LIN {X 0,Y 601.362,Z 589.903,A -85,B 0,C 180,E1 -618.877,E2 -618.877} C_VEL
LIN {X 0,Y 601.346,Z 594.511,A -85,B 0,C 180,E1 -619.903,E2 -619.903} C_VEL
LIN {X 0,Y 601.347,Z 599.168,A -85,B 0,C 180,E1 -621.261,E2 -621.261} C_VEL
LIN {X 0,Y 601.322,Z 602.306,A -85,B 0,C 180,E1 -622.613,E2 -622.613} C_VEL
LIN {X 0,Y 601.333,Z 604.045,A -85,B 0,C 180,E1 -623.962,E2 -623.962} C_VEL
LIN {X 0,Y 601.32,Z 604.445,A -85,B 0,C 180,E1 -625.307,E2 -625.307} C_VEL
LIN {X 0,Y 601.333,Z 603.522,A -85,B 0,C 180,E1 -626.65,E2 -626.65} C_VEL
LIN {X 0,Y 601.343,Z 601.262,A -85,B 0,C 180,E1 -627.991,E2 -627.991} C_VEL
LIN {X 0,Y 601.339,Z 597.609,A -85,B 0,C 180,E1 -629.33,E2 -629.33} C_VEL
LIN {X 0,Y 601.362,Z 592.469,A -85,B 0,C 180,E1 -630.67,E2 -630.67} C_VEL
LIN {X 0,Y 601.361,Z 587.493,A -85,B 0,C 180,E1 -631.674,E2 -631.674} C_VEL
LIN {X 0,Y 601.372,Z 580.4,A -85,B 0,C 180,E1 -632.847,E2 -632.847} C_VEL
LIN {X 0,Y 601.4,Z 571.651,A -85,B 0,C 180,E1 -634.021,E2 -634.021} C_VEL
LIN {X 0,Y 601.437,Z 562.527,A -85,B 0,C 180,E1 -635.028,E2 -635.028} C_VEL
LIN {X 0,Y 601.484,Z 552.47,A -85,B 0,C 180,E1 -635.952,E2 -635.952} C_VEL
LIN {X 0,Y 601.549,Z 541.565,A -85,B 0,C 180,E1 -636.785,E2 -636.785} C_VEL
LIN {X 0,Y 601.558,Z 529.313,A -85,B 0,C 180,E1 -637.552,E2 -637.552} C_VEL
LIN {X 0,Y 601.633,Z 515.778,A -85,B 0,C 180,E1 -638.227,E2 -638.227} C_VEL
LIN {X 0,Y 601.682,Z 502.635,A -85,B 0,C 180,E1 -638.734,E2 -638.734} C_VEL
LIN {X 0,Y 601.718,Z 488.359,A -85,B 0,C 180,E1 -639.136,E2 -639.136} C_VEL
LIN {X 0,Y 601.721,Z 474.417,A -85,B 0,C 180,E1 -639.39,E2 -639.39} C_VEL
LIN {X 0,Y 601.709,Z 344.001,A -85,B 0,C 180,E1 -640.974,E2 -640.974} C_VEL
LIN {X 0,Y 601.502,Z 342.735,A -85,B 0,C 180,E1 -640.998,E2 -640.998} C_VEL
LIN {X 0,Y 601.548,Z 324.422,A -85,B 0,C 180,E1 -643.666,E2 -643.666} C_VEL
LIN {X 0,Y 601.527,Z 310.251,A -85,B 0,C 180,E1 -645.762,E2 -645.762} C_VEL
LIN {X 0,Y 601.357,Z 309.2,A -85,B 0,C 180,E1 -645.941,E2 -645.941} C_VEL
LIN {X 0,Y 601.393,Z 309.2,A -85,B 0,C 180,E1 -648.811,E2 -648.811} C_VEL
LIN {X 0,Y 601.382,Z 309.199,A -85,B 0,C 180,E1 -651.24,E2 -651.24} C_VEL
LIN {X 0,Y 601.359,Z 309.199,A -85,B 0,C 180,E1 -653.413,E2 -653.413} C_VEL
LIN {X 0,Y 601.349,Z 309.198,A -85,B 0,C 180,E1 -655.854,E2 -655.854} C_VEL
LIN {X 0,Y 601.405,Z 309.197,A -85,B 0,C 180,E1 -658.628,E2 -658.628} C_VEL
LIN {X 0,Y 601.373,Z 309.194,A -85,B 0,C 180,E1 -661.729,E2 -661.729} C_VEL
LIN {X 0,Y 601.358,Z 309.197,A -85,B 0,C 180,E1 -664.123,E2 -664.123} C_VEL
LIN {X 0,Y 601.376,Z 309.202,A -85,B 0,C 180,E1 -666.585,E2 -666.585} C_VEL
LIN {X 0,Y 601.381,Z 309.194,A -85,B 0,C 180,E1 -669.528,E2 -669.528} C_VEL
LIN {X 0,Y 601.357,Z 309.196,A -85,B 0,C 180,E1 -671.771,E2 -671.771} C_VEL
LIN {X 0,Y 601.374,Z 309.203,A -85,B 0,C 180,E1 -674.53,E2 -674.53} C_VEL
LIN {X 0,Y 601.41,Z 309.197,A -85,B 0,C 180,E1 -676.43,E2 -676.43} C_VEL
LIN {X 0,Y 601.374,Z 309.197,A -85,B 0,C 180,E1 -679.122,E2 -679.122} C_VEL
LIN {X 0,Y 601.346,Z 309.198,A -85,B 0,C 180,E1 -681.726,E2 -681.726} C_VEL
LIN {X 0,Y 601.374,Z 309.2,A -85,B 0,C 180,E1 -684.244,E2 -684.244} C_VEL
LIN {X 0,Y 601.41,Z 309.197,A -85,B 0,C 180,E1 -686.685,E2 -686.685} C_VEL
LIN {X 0,Y 601.39,Z 309.194,A -85,B 0,C 180,E1 -689.056,E2 -689.056} C_VEL
LIN {X 0,Y 601.387,Z 309.192,A -85,B 0,C 180,E1 -691.37,E2 -691.37} C_VEL
LIN {X 0,Y 601.399,Z 309.197,A -85,B 0,C 180,E1 -694.136,E2 -694.136} C_VEL
LIN {X 0,Y 601.378,Z 309.2,A -85,B 0,C 180,E1 -696.588,E2 -696.588} C_VEL
LIN {X 0,Y 601.394,Z 309.191,A -85,B 0,C 180,E1 -699.477,E2 -699.477} C_VEL
LIN {X 0,Y 601.367,Z 309.195,A -85,B 0,C 180,E1 -701.606,E2 -701.606} C_VEL
LIN {X 0,Y 601.401,Z 309.199,A -85,B 0,C 180,E1 -704.408,E2 -704.408} C_VEL
LIN {X 0,Y 601.368,Z 309.194,A -85,B 0,C 180,E1 -707.17,E2 -707.17} C_VEL
LIN {X 0,Y 601.422,Z 309.192,A -85,B 0,C 180,E1 -709.905,E2 -709.905} C_VEL
LIN {X 0,Y 601.407,Z 309.194,A -85,B 0,C 180,E1 -712.614,E2 -712.614} C_VEL
LIN {X 0,Y 601.386,Z 309.193,A -85,B 0,C 180,E1 -715.307,E2 -715.307} C_VEL
LIN {X 0,Y 601.425,Z 309.196,A -85,B 0,C 180,E1 -717.991,E2 -717.991} C_VEL
LIN {X 0,Y 601.444,Z 309.187,A -85,B 0,C 180,E1 -720.669,E2 -720.669} C_VEL
LIN {X 0,Y 601.368,Z 309.196,A -85,B 0,C 180,E1 -723.35,E2 -723.35} C_VEL
LIN {X 0,Y 601.41,Z 309.2,A -85,B 0,C 180,E1 -726.037,E2 -726.037} C_VEL
LIN {X 0,Y 601.406,Z 309.191,A -85,B 0,C 180,E1 -728.738,E2 -728.738} C_VEL
LIN {X 0,Y 601.406,Z 309.193,A -85,B 0,C 180,E1 -731.459,E2 -731.459} C_VEL
LIN {X 0,Y 601.424,Z 309.193,A -85,B 0,C 180,E1 -734.205,E2 -734.205} C_VEL
LIN {X 0,Y 601.407,Z 309.19,A -85,B 0,C 180,E1 -736.986,E2 -736.986} C_VEL
LIN {X 0,Y 601.411,Z 309.19,A -85,B 0,C 180,E1 -739.099,E2 -739.099} C_VEL
LIN {X 0,Y 601.396,Z 309.193,A -85,B 0,C 180,E1 -741.24,E2 -741.24} C_VEL
LIN {X 0,Y 601.463,Z 309.188,A -85,B 0,C 180,E1 -744.14,E2 -744.14} C_VEL
LIN {X 0,Y 601.396,Z 309.193,A -85,B 0,C 180,E1 -747.114,E2 -747.114} C_VEL
LIN {X 0,Y 601.405,Z 309.195,A -85,B 0,C 180,E1 -749.394,E2 -749.394} C_VEL
LIN {X 0,Y 601.404,Z 309.201,A -85,B 0,C 180,E1 -751.727,E2 -751.727} C_VEL
LIN {X 0,Y 601.427,Z 309.191,A -85,B 0,C 180,E1 -754.118,E2 -754.118} C_VEL
LIN {X 0,Y 601.395,Z 309.192,A -85,B 0,C 180,E1 -756.583,E2 -756.583} C_VEL
LIN {X 0,Y 601.397,Z 309.194,A -85,B 0,C 180,E1 -759.128,E2 -759.128} C_VEL
LIN {X 0,Y 601.425,Z 309.195,A -85,B 0,C 180,E1 -761.765,E2 -761.765} C_VEL
LIN {X 0,Y 601.4,Z 309.191,A -85,B 0,C 180,E1 -764.532,E2 -764.532} C_VEL
LIN {X 0,Y 601.41,Z 309.199,A -85,B 0,C 180,E1 -767.41,E2 -767.41} C_VEL
LIN {X 0,Y 601.403,Z 309.193,A -85,B 0,C 180,E1 -770.004,E2 -770.004} C_VEL
LIN {X 0,Y 601.433,Z 309.187,A -85,B 0,C 180,E1 -772.618,E2 -772.618} C_VEL
LIN {X 0,Y 601.407,Z 309.195,A -85,B 0,C 180,E1 -775.067,E2 -775.067} C_VEL
LIN {X 0,Y 601.433,Z 309.196,A -85,B 0,C 180,E1 -777.484,E2 -777.484} C_VEL
LIN {X 0,Y 601.431,Z 309.19,A -85,B 0,C 180,E1 -779.851,E2 -779.851} C_VEL
LIN {X 0,Y 601.409,Z 309.191,A -85,B 0,C 180,E1 -782.639,E2 -782.639} C_VEL
LIN {X 0,Y 601.398,Z 309.2,A -85,B 0,C 180,E1 -785.121,E2 -785.121} C_VEL
LIN {X 0,Y 601.44,Z 309.309,A -85,B 0,C 180,E1 -786.179,E2 -786.179} C_VEL
LIN {X 0,Y 601.727,Z 314.043,A -85,B 0,C 180,E1 -786.803,E2 -786.803} C_VEL
LIN {X 0,Y 601.659,Z 335.098,A -85,B 0,C 180,E1 -789.486,E2 -789.486} C_VEL
LIN {X 0,Y 601.576,Z 357.707,A -85,B 0,C 180,E1 -792.317,E2 -792.317} C_VEL
LIN {X 0,Y 601.55,Z 371.484,A -85,B 0,C 180,E1 -794.021,E2 -794.021} C_VEL
LIN {X 0,Y 601.841,Z 375.607,A -85,B 0,C 180,E1 -794.094,E2 -794.094} C_VEL
LIN {X 0,Y 601.754,Z 508.902,A -85,B 0,C 180,E1 -795.72,E2 -795.72} C_VEL
LIN {X 0,Y 601.713,Z 523.291,A -85,B 0,C 180,E1 -796.029,E2 -796.029} C_VEL
LIN {X 0,Y 601.651,Z 537.71,A -85,B 0,C 180,E1 -796.489,E2 -796.489} C_VEL
LIN {X 0,Y 601.609,Z 551.632,A -85,B 0,C 180,E1 -797.09,E2 -797.09} C_VEL
LIN {X 0,Y 601.546,Z 564.092,A -85,B 0,C 180,E1 -797.775,E2 -797.775} C_VEL
LIN {X 0,Y 601.504,Z 575.471,A -85,B 0,C 180,E1 -798.543,E2 -798.543} C_VEL
LIN {X 0,Y 601.482,Z 585.931,A -85,B 0,C 180,E1 -799.395,E2 -799.395} C_VEL
LIN {X 0,Y 601.43,Z 596.333,A -85,B 0,C 180,E1 -800.415,E2 -800.415} C_VEL
LIN {X 0,Y 601.407,Z 604.913,A -85,B 0,C 180,E1 -801.431,E2 -801.431} C_VEL
LIN {X 0,Y 601.392,Z 613.114,A -85,B 0,C 180,E1 -802.614,E2 -802.614} C_VEL
LIN {X 0,Y 601.361,Z 618.751,A -85,B 0,C 180,E1 -803.604,E2 -803.604} C_VEL
LIN {X 0,Y 601.355,Z 623.568,A -85,B 0,C 180,E1 -804.635,E2 -804.635} C_VEL
LIN {X 0,Y 601.343,Z 628.442,A -85,B 0,C 180,E1 -805.979,E2 -805.979} C_VEL
LIN {X 0,Y 601.324,Z 631.831,A -85,B 0,C 180,E1 -807.32,E2 -807.32} C_VEL
LIN {X 0,Y 601.342,Z 633.831,A -85,B 0,C 180,E1 -808.661,E2 -808.661} C_VEL
LIN {X 0,Y 601.333,Z 634.5,A -85,B 0,C 180,E1 -810,E2 -810} C_VEL
LIN {X 0,Y 601.342,Z 633.831,A -85,B 0,C 180,E1 -811.339,E2 -811.339} C_VEL
LIN {X 0,Y 601.324,Z 631.831,A -85,B 0,C 180,E1 -812.68,E2 -812.68} C_VEL
LIN {X 0,Y 601.343,Z 628.442,A -85,B 0,C 180,E1 -814.021,E2 -814.021} C_VEL
LIN {X 0,Y 601.355,Z 623.567,A -85,B 0,C 180,E1 -815.365,E2 -815.365} C_VEL
LIN {X 0,Y 601.355,Z 617.051,A -85,B 0,C 180,E1 -816.712,E2 -816.712} C_VEL
LIN {X 0,Y 601.398,Z 609.797,A -85,B 0,C 180,E1 -817.892,E2 -817.892} C_VEL
LIN {X 0,Y 601.43,Z 600.822,A -85,B 0,C 180,E1 -819.077,E2 -819.077} C_VEL
LIN {X 0,Y 601.44,Z 591.39,A -85,B 0,C 180,E1 -820.095,E2 -820.095} C_VEL
LIN {X 0,Y 601.505,Z 580.693,A -85,B 0,C 180,E1 -821.05,E2 -821.05} C_VEL
LIN {X 0,Y 601.544,Z 569.425,A -85,B 0,C 180,E1 -821.883,E2 -821.883} C_VEL
LIN {X 0,Y 601.565,Z 556.641,A -85,B 0,C 180,E1 -822.654,E2 -822.654} C_VEL
LIN {X 0,Y 601.626,Z 544.155,A -85,B 0,C 180,E1 -823.253,E2 -823.253} C_VEL
LIN {X 0,Y 601.691,Z 530.829,A -85,B 0,C 180,E1 -823.749,E2 -823.749} C_VEL
LIN {X 0,Y 601.701,Z 517.407,A -85,B 0,C 180,E1 -824.114,E2 -824.114} C_VEL
LIN {X 0,Y 601.74,Z 503.82,A -85,B 0,C 180,E1 -824.353,E2 -824.353} C_VEL
LIN {X 0,Y 601.679,Z 372.472,A -85,B 0,C 180,E1 -825.948,E2 -825.948} C_VEL
LIN {X 0,Y 601.55,Z 371.484,A -85,B 0,C 180,E1 -825.979,E2 -825.979} C_VEL
LIN {X 0,Y 601.618,Z 348.143,A -85,B 0,C 180,E1 -828.874,E2 -828.874} C_VEL
LIN {X 0,Y 601.685,Z 326.619,A -85,B 0,C 180,E1 -831.589,E2 -831.589} C_VEL
LIN {X 0,Y 601.734,Z 311.075,A -85,B 0,C 180,E1 -833.58,E2 -833.58} C_VEL
LIN {X 0,Y 601.421,Z 309.193,A -85,B 0,C 180,E1 -833.867,E2 -833.867} C_VEL
LIN {X 0,Y 601.4,Z 309.197,A -85,B 0,C 180,E1 -836.364,E2 -836.364} C_VEL
LIN {X 0,Y 601.438,Z 309.195,A -85,B 0,C 180,E1 -838.789,E2 -838.789} C_VEL
LIN {X 0,Y 601.419,Z 309.189,A -85,B 0,C 180,E1 -841.454,E2 -841.454} C_VEL
LIN {X 0,Y 601.432,Z 309.19,A -85,B 0,C 180,E1 -844.118,E2 -844.118} C_VEL
LIN {X 0,Y 601.401,Z 309.202,A -85,B 0,C 180,E1 -846.583,E2 -846.583} C_VEL
LIN {X 0,Y 601.406,Z 309.192,A -85,B 0,C 180,E1 -849.127,E2 -849.127} C_VEL
LIN {X 0,Y 601.422,Z 309.189,A -85,B 0,C 180,E1 -851.766,E2 -851.766} C_VEL
LIN {X 0,Y 601.4,Z 309.2,A -85,B 0,C 180,E1 -854.533,E2 -854.533} C_VEL
LIN {X 0,Y 601.412,Z 309.189,A -85,B 0,C 180,E1 -857.41,E2 -857.41} C_VEL
LIN {X 0,Y 601.403,Z 309.195,A -85,B 0,C 180,E1 -860.004,E2 -860.004} C_VEL
LIN {X 0,Y 601.432,Z 309.193,A -85,B 0,C 180,E1 -862.619,E2 -862.619} C_VEL
LIN {X 0,Y 601.395,Z 309.192,A -85,B 0,C 180,E1 -865.067,E2 -865.067} C_VEL
LIN {X 0,Y 601.429,Z 309.188,A -85,B 0,C 180,E1 -867.484,E2 -867.484} C_VEL
LIN {X 0,Y 601.433,Z 309.19,A -85,B 0,C 180,E1 -869.852,E2 -869.852} C_VEL
LIN {X 0,Y 601.39,Z 309.196,A -85,B 0,C 180,E1 -872.643,E2 -872.643} C_VEL
LIN {X 0,Y 601.391,Z 309.192,A -85,B 0,C 180,E1 -875.121,E2 -875.121} C_VEL
LIN {X 0,Y 601.419,Z 309.189,A -85,B 0,C 180,E1 -877.395,E2 -877.395} C_VEL
LIN {X 0,Y 601.398,Z 309.201,A -85,B 0,C 180,E1 -880.19,E2 -880.19} C_VEL
LIN {X 0,Y 601.387,Z 309.199,A -85,B 0,C 180,E1 -882.311,E2 -882.311} C_VEL
LIN {X 0,Y 601.398,Z 309.196,A -85,B 0,C 180,E1 -884.408,E2 -884.408} C_VEL
LIN {X 0,Y 601.405,Z 309.19,A -85,B 0,C 180,E1 -887.172,E2 -887.172} C_VEL
LIN {X 0,Y 601.431,Z 309.196,A -85,B 0,C 180,E1 -889.905,E2 -889.905} C_VEL
LIN {X 0,Y 601.38,Z 309.195,A -85,B 0,C 180,E1 -892.614,E2 -892.614} C_VEL
LIN {X 0,Y 601.417,Z 309.19,A -85,B 0,C 180,E1 -895.308,E2 -895.308} C_VEL
LIN {X 0,Y 601.424,Z 309.197,A -85,B 0,C 180,E1 -897.991,E2 -897.991} C_VEL
LIN {X 0,Y 601.442,Z 309.194,A -85,B 0,C 180,E1 -900,E2 -900} C_VEL
LIN {X 0,Y 601.407,Z 309.19,A -85,B 0,C 180,E1 -902.679,E2 -902.679} C_VEL
LIN {X 0,Y 601.418,Z 309.192,A -85,B 0,C 180,E1 -905.364,E2 -905.364} C_VEL
LIN {X 0,Y 601.409,Z 309.196,A -85,B 0,C 180,E1 -908.061,E2 -908.061} C_VEL
LIN {X 0,Y 601.402,Z 309.191,A -85,B 0,C 180,E1 -910.998,E2 -910.998} C_VEL
LIN {X 0,Y 601.38,Z 309.195,A -85,B 0,C 180,E1 -912.33,E2 -912.33} C_VEL
LIN {X 0,Y 600.695,Z 309.281,A -85,B 0,C 180,E1 -912.89,E2 -912.89} C_VEL
LIN {X 0,Y 597.844,Z 309.643,A -85,B 0,C 180,E1 -913.797,E2 -913.797} C_VEL
LIN {X 0,Y 595.447,Z 309.937,A -85,B 0,C 180,E1 -914.528,E2 -914.528} C_VEL
LIN {X 0,Y 594.418,Z 310.063,A -85,B 0,C 180,E1 -915.091,E2 -915.091} C_VEL
LIN {X 0,Y 594.333,Z 310.074,A -85,B 0,C 180,E1 -915.282,E2 -915.282} C_VEL
LIN {X 0,Y 594.328,Z 310.078,A -85,B 0,C 180,E1 -917.906,E2 -917.906} C_VEL
LIN {X 0,Y 594.375,Z 310.066,A -85,B 0,C 180,E1 -920.777,E2 -920.777} C_VEL
LIN {X 0,Y 594.345,Z 310.078,A -85,B 0,C 180,E1 -923.706,E2 -923.706} C_VEL
LIN {X 0,Y 594.354,Z 310.072,A -85,B 0,C 180,E1 -926.015,E2 -926.015} C_VEL
LIN {X 0,Y 594.343,Z 310.072,A -85,B 0,C 180,E1 -928.95,E2 -928.95} C_VEL
LIN {X 0,Y 594.359,Z 310.076,A -85,B 0,C 180,E1 -931.639,E2 -931.639} C_VEL
LIN {X 0,Y 594.354,Z 310.069,A -85,B 0,C 180,E1 -934.582,E2 -934.582} C_VEL
LIN {X 0,Y 594.356,Z 310.076,A -85,B 0,C 180,E1 -937.604,E2 -937.604} C_VEL
LIN {X 0,Y 594.317,Z 310.074,A -85,B 0,C 180,E1 -940.572,E2 -940.572} C_VEL
LIN {X 0,Y 594.342,Z 310.08,A -85,B 0,C 180,E1 -943.302,E2 -943.302} C_VEL
LIN {X 0,Y 594.316,Z 310.073,A -85,B 0,C 180,E1 -946.166,E2 -946.166} C_VEL
LIN {X 0,Y 594.322,Z 310.074,A -85,B 0,C 180,E1 -948.531,E2 -948.531} C_VEL
LIN {X 0,Y 594.325,Z 310.082,A -85,B 0,C 180,E1 -951.303,E2 -951.303} C_VEL
LIN {X 0,Y 594.311,Z 310.077,A -85,B 0,C 180,E1 -953.752,E2 -953.752} C_VEL
LIN {X 0,Y 594.318,Z 310.073,A -85,B 0,C 180,E1 -956.235,E2 -956.235} C_VEL
LIN {X 0,Y 594.339,Z 310.074,A -85,B 0,C 180,E1 -958.648,E2 -958.648} C_VEL
LIN {X 0,Y 594.345,Z 310.08,A -85,B 0,C 180,E1 -961.05,E2 -961.05} C_VEL
LIN {X 0,Y 594.349,Z 310.079,A -85,B 0,C 180,E1 -963.299,E2 -963.299} C_VEL
LIN {X 0,Y 594.343,Z 310.174,A -85,B 0,C 180,E1 -964.054,E2 -964.054} C_VEL
LIN {X 0,Y 594.621,Z 316.43,A -85,B 0,C 180,E1 -965.005,E2 -965.005} C_VEL
LIN {X 0,Y 594.526,Z 335.069,A -85,B 0,C 180,E1 -967.773,E2 -967.773} C_VEL
LIN {X 0,Y 594.505,Z 342.736,A -85,B 0,C 180,E1 -968.9,E2 -968.9} C_VEL
LIN {X 0,Y 595.013,Z 346.636,A -85,B 0,C 180,E1 -968.964,E2 -968.964} C_VEL
LIN {X 0,Y 594.868,Z 479.926,A -85,B 0,C 180,E1 -970.615,E2 -970.615} C_VEL
LIN {X 0,Y 594.81,Z 494.165,A -85,B 0,C 180,E1 -970.934,E2 -970.934} C_VEL
LIN {X 0,Y 594.725,Z 508.209,A -85,B 0,C 180,E1 -971.393,E2 -971.393} C_VEL
LIN {X 0,Y 594.641,Z 522.314,A -85,B 0,C 180,E1 -972.015,E2 -972.015} C_VEL
LIN {X 0,Y 594.59,Z 534.903,A -85,B 0,C 180,E1 -972.724,E2 -972.724} C_VEL
LIN {X 0,Y 594.494,Z 546.361,A -85,B 0,C 180,E1 -973.517,E2 -973.517} C_VEL
LIN {X 0,Y 594.459,Z 556.875,A -85,B 0,C 180,E1 -974.397,E2 -974.397} C_VEL
LIN {X 0,Y 594.382,Z 567.253,A -85,B 0,C 180,E1 -975.448,E2 -975.448} C_VEL
LIN {X 0,Y 594.342,Z 575.804,A -85,B 0,C 180,E1 -976.494,E2 -976.494} C_VEL
LIN {X 0,Y 594.291,Z 583.937,A -85,B 0,C 180,E1 -977.71,E2 -977.71} C_VEL
LIN {X 0,Y 594.252,Z 590.822,A -85,B 0,C 180,E1 -978.997,E2 -978.997} C_VEL
LIN {X 0,Y 594.26,Z 595.579,A -85,B 0,C 180,E1 -980.126,E2 -980.126} C_VEL
LIN {X 0,Y 594.247,Z 599,A -85,B 0,C 180,E1 -981.156,E2 -981.156} C_VEL
LIN {X 0,Y 594.248,Z 602.207,A -85,B 0,C 180,E1 -982.525,E2 -982.525} C_VEL
LIN {X 0,Y 594.238,Z 604.004,A -85,B 0,C 180,E1 -983.89,E2 -983.89} C_VEL
LIN {X 0,Y 594.219,Z 604.459,A -85,B 0,C 180,E1 -985.251,E2 -985.251} C_VEL
LIN {X 0,Y 594.253,Z 603.59,A -85,B 0,C 180,E1 -986.61,E2 -986.61} C_VEL
LIN {X 0,Y 594.241,Z 601.388,A -85,B 0,C 180,E1 -987.967,E2 -987.967} C_VEL
LIN {X 0,Y 594.241,Z 597.794,A -85,B 0,C 180,E1 -989.322,E2 -989.322} C_VEL
LIN {X 0,Y 594.267,Z 592.717,A -85,B 0,C 180,E1 -990.678,E2 -990.678} C_VEL
LIN {X 0,Y 594.284,Z 587.81,A -85,B 0,C 180,E1 -991.694,E2 -991.694} C_VEL
LIN {X 0,Y 594.303,Z 580.79,A -85,B 0,C 180,E1 -992.881,E2 -992.881} C_VEL
LIN {X 0,Y 594.347,Z 572.125,A -85,B 0,C 180,E1 -994.068,E2 -994.068} C_VEL
LIN {X 0,Y 594.387,Z 563.093,A -85,B 0,C 180,E1 -995.088,E2 -995.088} C_VEL
LIN {X 0,Y 594.494,Z 552.164,A -85,B 0,C 180,E1 -996.108,E2 -996.108} C_VEL
LIN {X 0,Y 594.579,Z 540.293,A -85,B 0,C 180,E1 -997.011,E2 -997.011} C_VEL
LIN {X 0,Y 594.611,Z 527.31,A -85,B 0,C 180,E1 -997.812,E2 -997.812} C_VEL
LIN {X 0,Y 594.688,Z 515.203,A -85,B 0,C 180,E1 -998.41,E2 -998.41} C_VEL
LIN {X 0,Y 594.799,Z 501.866,A -85,B 0,C 180,E1 -998.922,E2 -998.922} C_VEL
LIN {X 0,Y 594.845,Z 488.169,A -85,B 0,C 180,E1 -999.307,E2 -999.307} C_VEL
LIN {X 0,Y 594.867,Z 474.096,A -85,B 0,C 180,E1 -999.564,E2 -999.564} C_VEL
LIN {X 0,Y 594.981,Z 345.443,A -85,B 0,C 180,E1 -1001.141,E2 -1001.141} C_VEL
LIN {X 0,Y 594.487,Z 342.62,A -85,B 0,C 180,E1 -1001.208,E2 -1001.208} C_VEL
LIN {X 0,Y 594.557,Z 324.037,A -85,B 0,C 180,E1 -1003.951,E2 -1003.951} C_VEL
LIN {X 0,Y 594.595,Z 311.845,A -85,B 0,C 180,E1 -1005.775,E2 -1005.775} C_VEL
LIN {X 0,Y 594.346,Z 310.075,A -85,B 0,C 180,E1 -1006.09,E2 -1006.09} C_VEL
LIN {X 0,Y 594.349,Z 310.075,A -85,B 0,C 180,E1 -1009.335,E2 -1009.335} C_VEL
LIN {X 0,Y 594.337,Z 310.073,A -85,B 0,C 180,E1 -1011.505,E2 -1011.505} C_VEL
LIN {X 0,Y 594.328,Z 310.073,A -85,B 0,C 180,E1 -1013.707,E2 -1013.707} C_VEL
LIN {X 0,Y 594.347,Z 310.077,A -85,B 0,C 180,E1 -1016.702,E2 -1016.702} C_VEL
LIN {X 0,Y 594.312,Z 310.074,A -85,B 0,C 180,E1 -1019.78,E2 -1019.78} C_VEL
LIN {X 0,Y 594.341,Z 310.072,A -85,B 0,C 180,E1 -1022.149,E2 -1022.149} C_VEL
LIN {X 0,Y 594.318,Z 310.075,A -85,B 0,C 180,E1 -1025.318,E2 -1025.318} C_VEL
LIN {X 0,Y 594.302,Z 310.076,A -85,B 0,C 180,E1 -1027.947,E2 -1027.947} C_VEL
LIN {X 0,Y 594.358,Z 310.077,A -85,B 0,C 180,E1 -1030.819,E2 -1030.819} C_VEL
LIN {X 0,Y 594.317,Z 310.074,A -85,B 0,C 180,E1 -1033.834,E2 -1033.834} C_VEL
LIN {X 0,Y 594.342,Z 310.08,A -85,B 0,C 180,E1 -1036.698,E2 -1036.698} C_VEL
LIN {X 0,Y 594.317,Z 310.073,A -85,B 0,C 180,E1 -1039.428,E2 -1039.428} C_VEL
LIN {X 0,Y 594.356,Z 310.076,A -85,B 0,C 180,E1 -1042.396,E2 -1042.396} C_VEL
LIN {X 0,Y 594.355,Z 310.069,A -85,B 0,C 180,E1 -1045.418,E2 -1045.418} C_VEL
LIN {X 0,Y 594.368,Z 310.075,A -85,B 0,C 180,E1 -1048.36,E2 -1048.36} C_VEL
LIN {X 0,Y 594.343,Z 310.072,A -85,B 0,C 180,E1 -1051.05,E2 -1051.05} C_VEL
LIN {X 0,Y 594.361,Z 310.072,A -85,B 0,C 180,E1 -1054.055,E2 -1054.055} C_VEL
LIN {X 0,Y 594.347,Z 310.079,A -85,B 0,C 180,E1 -1056.294,E2 -1056.294} C_VEL
LIN {X 0,Y 594.376,Z 310.065,A -85,B 0,C 180,E1 -1059.223,E2 -1059.223} C_VEL
LIN {X 0,Y 594.329,Z 310.078,A -85,B 0,C 180,E1 -1062.094,E2 -1062.094} C_VEL
LIN {X 0,Y 594.342,Z 310.071,A -85,B 0,C 180,E1 -1064.921,E2 -1064.921} C_VEL
LIN {X 0,Y 594.349,Z 310.071,A -85,B 0,C 180,E1 -1067.711,E2 -1067.711} C_VEL
LIN {X 0,Y 594.358,Z 310.074,A -85,B 0,C 180,E1 -1070.471,E2 -1070.471} C_VEL
LIN {X 0,Y 594.367,Z 310.067,A -85,B 0,C 180,E1 -1073.34,E2 -1073.34} C_VEL
LIN {X 0,Y 594.349,Z 310.076,A -85,B 0,C 180,E1 -1075.931,E2 -1075.931} C_VEL
LIN {X 0,Y 594.371,Z 310.069,A -85,B 0,C 180,E1 -1078.645,E2 -1078.645} C_VEL
LIN {X 0,Y 594.415,Z 310.062,A -85,B 0,C 180,E1 -1080.677,E2 -1080.677} C_VEL
LIN {X 0,Y 594.323,Z 310.074,A -85,B 0,C 180,E1 -1083.389,E2 -1083.389} C_VEL
LIN {X 0,Y 594.367,Z 310.069,A -85,B 0,C 180,E1 -1085.428,E2 -1085.428} C_VEL
LIN {X 0,Y 594.383,Z 310.073,A -85,B 0,C 180,E1 -1088.157,E2 -1088.157} C_VEL
LIN {X 0,Y 594.374,Z 310.066,A -85,B 0,C 180,E1 -1091.063,E2 -1091.063} C_VEL
LIN {X 0,Y 594.373,Z 310.073,A -85,B 0,C 180,E1 -1093.679,E2 -1093.679} C_VEL
LIN {X 0,Y 594.377,Z 310.066,A -85,B 0,C 180,E1 -1096.712,E2 -1096.712} C_VEL
LIN {X 0,Y 594.363,Z 310.07,A -85,B 0,C 180,E1 -1099.334,E2 -1099.334} C_VEL
LIN {X 0,Y 594.36,Z 310.073,A -85,B 0,C 180,E1 -1101.503,E2 -1101.503} C_VEL
LIN {X 0,Y 594.393,Z 310.065,A -85,B 0,C 180,E1 -1104.446,E2 -1104.446} C_VEL
LIN {X 0,Y 594.361,Z 310.068,A -85,B 0,C 180,E1 -1106.701,E2 -1106.701} C_VEL
LIN {X 0,Y 594.378,Z 310.066,A -85,B 0,C 180,E1 -1108.999,E2 -1108.999} C_VEL
LIN {X 0,Y 594.379,Z 310.076,A -85,B 0,C 180,E1 -1111.642,E2 -1111.642} C_VEL
LIN {X 0,Y 594.373,Z 310.067,A -85,B 0,C 180,E1 -1114.58,E2 -1114.58} C_VEL
LIN {X 0,Y 594.388,Z 310.075,A -85,B 0,C 180,E1 -1117.608,E2 -1117.608} C_VEL
LIN {X 0,Y 594.365,Z 310.067,A -85,B 0,C 180,E1 -1120.567,E2 -1120.567} C_VEL
LIN {X 0,Y 594.367,Z 310.073,A -85,B 0,C 180,E1 -1123.299,E2 -1123.299} C_VEL
LIN {X 0,Y 594.361,Z 310.069,A -85,B 0,C 180,E1 -1126.161,E2 -1126.161} C_VEL
LIN {X 0,Y 594.376,Z 310.066,A -85,B 0,C 180,E1 -1128.535,E2 -1128.535} C_VEL
LIN {X 0,Y 594.381,Z 310.073,A -85,B 0,C 180,E1 -1131.296,E2 -1131.296} C_VEL
LIN {X 0,Y 594.396,Z 310.069,A -85,B 0,C 180,E1 -1133.758,E2 -1133.758} C_VEL
LIN {X 0,Y 594.377,Z 310.067,A -85,B 0,C 180,E1 -1136.238,E2 -1136.238} C_VEL
LIN {X 0,Y 594.369,Z 310.068,A -85,B 0,C 180,E1 -1138.649,E2 -1138.649} C_VEL
LIN {X 0,Y 594.385,Z 310.071,A -85,B 0,C 180,E1 -1141.042,E2 -1141.042} C_VEL
LIN {X 0,Y 594.385,Z 310.067,A -85,B 0,C 180,E1 -1143.978,E2 -1143.978} C_VEL
LIN {X 0,Y 594.427,Z 310.192,A -85,B 0,C 180,E1 -1145.996,E2 -1145.996} C_VEL
LIN {X 0,Y 594.847,Z 313.901,A -85,B 0,C 180,E1 -1146.5,E2 -1146.5} C_VEL
LIN {X 0,Y 594.771,Z 333.13,A -85,B 0,C 180,E1 -1148.986,E2 -1148.986} C_VEL
LIN {X 0,Y 594.649,Z 356.294,A -85,B 0,C 180,E1 -1151.926,E2 -1151.926} C_VEL
LIN {X 0,Y 594.541,Z 371.572,A -85,B 0,C 180,E1 -1153.838,E2 -1153.838} C_VEL
LIN {X 0,Y 595.026,Z 375.607,A -85,B 0,C 180,E1 -1153.907,E2 -1153.907} C_VEL
LIN {X 0,Y 594.876,Z 509.881,A -85,B 0,C 180,E1 -1155.569,E2 -1155.569} C_VEL
LIN {X 0,Y 594.816,Z 524.128,A -85,B 0,C 180,E1 -1155.888,E2 -1155.888} C_VEL
LIN {X 0,Y 594.74,Z 537.712,A -85,B 0,C 180,E1 -1156.329,E2 -1156.329} C_VEL
LIN {X 0,Y 594.663,Z 551.634,A -85,B 0,C 180,E1 -1156.937,E2 -1156.937} C_VEL
LIN {X 0,Y 594.581,Z 564.094,A -85,B 0,C 180,E1 -1157.629,E2 -1157.629} C_VEL
LIN {X 0,Y 594.524,Z 576.553,A -85,B 0,C 180,E1 -1158.487,E2 -1158.487} C_VEL
LIN {X 0,Y 594.449,Z 587.836,A -85,B 0,C 180,E1 -1159.441,E2 -1159.441} C_VEL
LIN {X 0,Y 594.368,Z 597.85,A -85,B 0,C 180,E1 -1160.471,E2 -1160.471} C_VEL
LIN {X 0,Y 594.323,Z 606.17,A -85,B 0,C 180,E1 -1161.5,E2 -1161.5} C_VEL
LIN {X 0,Y 594.303,Z 614.125,A -85,B 0,C 180,E1 -1162.696,E2 -1162.696} C_VEL
LIN {X 0,Y 594.279,Z 620.527,A -85,B 0,C 180,E1 -1163.89,E2 -1163.89} C_VEL
LIN {X 0,Y 594.237,Z 626.199,A -85,B 0,C 180,E1 -1165.251,E2 -1165.251} C_VEL
LIN {X 0,Y 594.259,Z 630.315,A -85,B 0,C 180,E1 -1166.61,E2 -1166.61} C_VEL
LIN {X 0,Y 594.24,Z 633,A -85,B 0,C 180,E1 -1167.967,E2 -1167.967} C_VEL
LIN {X 0,Y 594.237,Z 634.332,A -85,B 0,C 180,E1 -1169.322,E2 -1169.322} C_VEL
LIN {X 0,Y 594.237,Z 634.332,A -85,B 0,C 180,E1 -1170.678,E2 -1170.678} C_VEL
LIN {X 0,Y 594.24,Z 633,A -85,B 0,C 180,E1 -1172.033,E2 -1172.033} C_VEL
LIN {X 0,Y 594.259,Z 630.316,A -85,B 0,C 180,E1 -1173.39,E2 -1173.39} C_VEL
LIN {X 0,Y 594.237,Z 626.199,A -85,B 0,C 180,E1 -1174.749,E2 -1174.749} C_VEL
LIN {X 0,Y 594.279,Z 620.526,A -85,B 0,C 180,E1 -1176.11,E2 -1176.11} C_VEL
LIN {X 0,Y 594.303,Z 614.125,A -85,B 0,C 180,E1 -1177.304,E2 -1177.304} C_VEL
LIN {X 0,Y 594.324,Z 606.169,A -85,B 0,C 180,E1 -1178.5,E2 -1178.5} C_VEL
LIN {X 0,Y 594.367,Z 597.849,A -85,B 0,C 180,E1 -1179.529,E2 -1179.529} C_VEL
LIN {X 0,Y 594.449,Z 587.835,A -85,B 0,C 180,E1 -1180.559,E2 -1180.559} C_VEL
LIN {X 0,Y 594.524,Z 576.56,A -85,B 0,C 180,E1 -1181.512,E2 -1181.512} C_VEL
LIN {X 0,Y 594.582,Z 564.094,A -85,B 0,C 180,E1 -1182.371,E2 -1182.371} C_VEL
LIN {X 0,Y 594.663,Z 551.634,A -85,B 0,C 180,E1 -1183.063,E2 -1183.063} C_VEL
LIN {X 0,Y 594.74,Z 537.707,A -85,B 0,C 180,E1 -1183.671,E2 -1183.671} C_VEL
LIN {X 0,Y 594.816,Z 524.123,A -85,B 0,C 180,E1 -1184.112,E2 -1184.112} C_VEL
LIN {X 0,Y 594.859,Z 509.876,A -85,B 0,C 180,E1 -1184.431,E2 -1184.431} C_VEL
LIN {X 0,Y 594.933,Z 373.814,A -85,B 0,C 180,E1 -1186.118,E2 -1186.118} C_VEL
LIN {X 0,Y 594.551,Z 371.484,A -85,B 0,C 180,E1 -1186.172,E2 -1186.172} C_VEL
LIN {X 0,Y 594.677,Z 348.115,A -85,B 0,C 180,E1 -1189.107,E2 -1189.107} C_VEL
LIN {X 0,Y 594.792,Z 326.619,A -85,B 0,C 180,E1 -1191.852,E2 -1191.852} C_VEL
LIN {X 0,Y 594.825,Z 312.488,A -85,B 0,C 180,E1 -1193.686,E2 -1193.686} C_VEL
LIN {X 0,Y 594.4,Z 310.07,A -85,B 0,C 180,E1 -1194.028,E2 -1194.028} C_VEL
LIN {X 0,Y 594.38,Z 310.076,A -85,B 0,C 180,E1 -1196.7,E2 -1196.7} C_VEL
LIN {X 0,Y 594.384,Z 310.07,A -85,B 0,C 180,E1 -1198.999,E2 -1198.999} C_VEL
LIN {X 0,Y 594.378,Z 310.066,A -85,B 0,C 180,E1 -1201.643,E2 -1201.643} C_VEL
LIN {X 0,Y 594.381,Z 310.076,A -85,B 0,C 180,E1 -1204.58,E2 -1204.58} C_VEL
LIN {X 0,Y 594.389,Z 310.065,A -85,B 0,C 180,E1 -1207.608,E2 -1207.608} C_VEL
LIN {X 0,Y 594.369,Z 310.077,A -85,B 0,C 180,E1 -1210.567,E2 -1210.567} C_VEL
LIN {X 0,Y 594.366,Z 310.067,A -85,B 0,C 180,E1 -1213.3,E2 -1213.3} C_VEL
LIN {X 0,Y 594.362,Z 310.073,A -85,B 0,C 180,E1 -1216.162,E2 -1216.162} C_VEL
LIN {X 0,Y 594.378,Z 310.074,A -85,B 0,C 180,E1 -1218.536,E2 -1218.536} C_VEL
LIN {X 0,Y 594.372,Z 310.066,A -85,B 0,C 180,E1 -1221.298,E2 -1221.298} C_VEL
LIN {X 0,Y 594.352,Z 310.071,A -85,B 0,C 180,E1 -1223.756,E2 -1223.756} C_VEL
LIN {X 0,Y 594.377,Z 310.075,A -85,B 0,C 180,E1 -1226.239,E2 -1226.239} C_VEL
LIN {X 0,Y 594.368,Z 310.071,A -85,B 0,C 180,E1 -1228.65,E2 -1228.65} C_VEL
LIN {X 0,Y 594.381,Z 310.066,A -85,B 0,C 180,E1 -1231.044,E2 -1231.044} C_VEL
LIN {X 0,Y 594.375,Z 310.074,A -85,B 0,C 180,E1 -1234.056,E2 -1234.056} C_VEL
LIN {X 0,Y 594.375,Z 310.075,A -85,B 0,C 180,E1 -1236.295,E2 -1236.295} C_VEL
LIN {X 0,Y 594.399,Z 310.063,A -85,B 0,C 180,E1 -1239.224,E2 -1239.224} C_VEL
LIN {X 0,Y 594.349,Z 310.079,A -85,B 0,C 180,E1 -1242.095,E2 -1242.095} C_VEL
LIN {X 0,Y 594.357,Z 310.077,A -85,B 0,C 180,E1 -1244.219,E2 -1244.219} C_VEL
LIN {X 0,Y 594.373,Z 310.072,A -85,B 0,C 180,E1 -1246.321,E2 -1246.321} C_VEL
LIN {X 0,Y 594.354,Z 310.069,A -85,B 0,C 180,E1 -1249.094,E2 -1249.094} C_VEL
LIN {X 0,Y 594.384,Z 310.073,A -85,B 0,C 180,E1 -1251.843,E2 -1251.843} C_VEL
LIN {X 0,Y 594.366,Z 310.069,A -85,B 0,C 180,E1 -1254.572,E2 -1254.572} C_VEL
LIN {X 0,Y 594.399,Z 310.064,A -85,B 0,C 180,E1 -1257.289,E2 -1257.289} C_VEL
LIN {X 0,Y 594.411,Z 310.07,A -85,B 0,C 180,E1 -1260,E2 -1260} C_VEL
LIN {X 0,Y 594.377,Z 310.066,A -85,B 0,C 180,E1 -1262.711,E2 -1262.711} C_VEL
LIN {X 0,Y 594.383,Z 310.069,A -85,B 0,C 180,E1 -1265.428,E2 -1265.428} C_VEL
LIN {X 0,Y 594.358,Z 310.072,A -85,B 0,C 180,E1 -1268.158,E2 -1268.158} C_VEL
LIN {X 0,Y 594.369,Z 310.068,A -85,B 0,C 180,E1 -1271.061,E2 -1271.061} C_VEL
LIN {X 0,Y 594.359,Z 310.071,A -85,B 0,C 180,E1 -1274.16,E2 -1274.16} C_VEL
LIN {X 0,Y 594.333,Z 310.074,A -85,B 0,C 180,E1 -1275.282,E2 -1275.282} C_VEL
LIN {X 0,Y 593.661,Z 310.164,A -85,B 0,C 180,E1 -1275.848,E2 -1275.848} C_VEL
LIN {X 0,Y 590.795,Z 310.521,A -85,B 0,C 180,E1 -1276.765,E2 -1276.765} C_VEL
LIN {X 0,Y 588.383,Z 310.819,A -85,B 0,C 180,E1 -1277.503,E2 -1277.503} C_VEL
LIN {X 0,Y 587.358,Z 310.944,A -85,B 0,C 180,E1 -1278.073,E2 -1278.073} C_VEL
LIN {X 0,Y 587.281,Z 310.952,A -85,B 0,C 180,E1 -1278.266,E2 -1278.266} C_VEL
LIN {X 0,Y 587.302,Z 310.948,A -85,B 0,C 180,E1 -1281.039,E2 -1281.039} C_VEL
LIN {X 0,Y 587.285,Z 310.952,A -85,B 0,C 180,E1 -1284.009,E2 -1284.009} C_VEL
LIN {X 0,Y 587.3,Z 310.948,A -85,B 0,C 180,E1 -1286.281,E2 -1286.281} C_VEL
LIN {X 0,Y 587.303,Z 310.951,A -85,B 0,C 180,E1 -1289.124,E2 -1289.124} C_VEL
LIN {X 0,Y 587.319,Z 310.95,A -85,B 0,C 180,E1 -1291.831,E2 -1291.831} C_VEL
LIN {X 0,Y 587.325,Z 310.944,A -85,B 0,C 180,E1 -1294.344,E2 -1294.344} C_VEL
LIN {X 0,Y 587.31,Z 310.953,A -85,B 0,C 180,E1 -1297.611,E2 -1297.611} C_VEL
LIN {X 0,Y 587.277,Z 310.95,A -85,B 0,C 180,E1 -1300.258,E2 -1300.258} C_VEL
LIN {X 0,Y 587.283,Z 310.956,A -85,B 0,C 180,E1 -1303.114,E2 -1303.114} C_VEL
LIN {X 0,Y 587.272,Z 310.951,A -85,B 0,C 180,E1 -1306.044,E2 -1306.044} C_VEL
LIN {X 0,Y 587.269,Z 310.957,A -85,B 0,C 180,E1 -1308.933,E2 -1308.933} C_VEL
LIN {X 0,Y 587.271,Z 310.957,A -85,B 0,C 180,E1 -1311.516,E2 -1311.516} C_VEL
LIN {X 0,Y 587.257,Z 310.953,A -85,B 0,C 180,E1 -1314.097,E2 -1314.097} C_VEL
LIN {X 0,Y 587.292,Z 310.951,A -85,B 0,C 180,E1 -1316.6,E2 -1316.6} C_VEL
LIN {X 0,Y 587.289,Z 310.954,A -85,B 0,C 180,E1 -1319.499,E2 -1319.499} C_VEL
LIN {X 0,Y 587.3,Z 310.95,A -85,B 0,C 180,E1 -1322.318,E2 -1322.318} C_VEL
LIN {X 0,Y 587.325,Z 311.083,A -85,B 0,C 180,E1 -1323.93,E2 -1323.93} C_VEL
LIN {X 0,Y 587.673,Z 317.221,A -85,B 0,C 180,E1 -1324.878,E2 -1324.878} C_VEL
LIN {X 0,Y 587.53,Z 335.863,A -85,B 0,C 180,E1 -1327.679,E2 -1327.679} C_VEL
LIN {X 0,Y 587.544,Z 342.992,A -85,B 0,C 180,E1 -1328.709,E2 -1328.709} C_VEL
LIN {X 0,Y 588.214,Z 347.161,A -85,B 0,C 180,E1 -1328.78,E2 -1328.78} C_VEL
LIN {X 0,Y 587.994,Z 478.945,A -85,B 0,C 180,E1 -1330.425,E2 -1330.425} C_VEL
LIN {X 0,Y 587.93,Z 493.225,A -85,B 0,C 180,E1 -1330.738,E2 -1330.738} C_VEL
LIN {X 0,Y 587.832,Z 506.593,A -85,B 0,C 180,E1 -1331.167,E2 -1331.167} C_VEL
LIN {X 0,Y 587.775,Z 519.267,A -85,B 0,C 180,E1 -1331.707,E2 -1331.707} C_VEL
LIN {X 0,Y 587.634,Z 532.446,A -85,B 0,C 180,E1 -1332.423,E2 -1332.423} C_VEL
LIN {X 0,Y 587.537,Z 544.443,A -85,B 0,C 180,E1 -1333.234,E2 -1333.234} C_VEL
LIN {X 0,Y 587.453,Z 556.182,A -85,B 0,C 180,E1 -1334.206,E2 -1334.206} C_VEL
LIN {X 0,Y 587.358,Z 566.717,A -85,B 0,C 180,E1 -1335.27,E2 -1335.27} C_VEL
LIN {X 0,Y 587.284,Z 575.362,A -85,B 0,C 180,E1 -1336.329,E2 -1336.329} C_VEL
LIN {X 0,Y 587.218,Z 583.578,A -85,B 0,C 180,E1 -1337.559,E2 -1337.559} C_VEL
LIN {X 0,Y 587.203,Z 589.347,A -85,B 0,C 180,E1 -1338.61,E2 -1338.61} C_VEL
LIN {X 0,Y 587.177,Z 594.008,A -85,B 0,C 180,E1 -1339.657,E2 -1339.657} C_VEL
LIN {X 0,Y 587.152,Z 598.817,A -85,B 0,C 180,E1 -1341.048,E2 -1341.048} C_VEL
LIN {X 0,Y 587.147,Z 602.103,A -85,B 0,C 180,E1 -1342.434,E2 -1342.434} C_VEL
LIN {X 0,Y 587.148,Z 603.961,A -85,B 0,C 180,E1 -1343.816,E2 -1343.816} C_VEL
LIN {X 0,Y 587.119,Z 604.472,A -85,B 0,C 180,E1 -1345.193,E2 -1345.193} C_VEL
LIN {X 0,Y 587.177,Z 603.659,A -85,B 0,C 180,E1 -1346.569,E2 -1346.569} C_VEL
LIN {X 0,Y 587.14,Z 601.513,A -85,B 0,C 180,E1 -1347.942,E2 -1347.942} C_VEL
LIN {X 0,Y 587.143,Z 597.979,A -85,B 0,C 180,E1 -1349.314,E2 -1349.314} C_VEL
LIN {X 0,Y 587.173,Z 592.965,A -85,B 0,C 180,E1 -1350.686,E2 -1350.686} C_VEL
LIN {X 0,Y 587.208,Z 586.323,A -85,B 0,C 180,E1 -1352.058,E2 -1352.058} C_VEL
LIN {X 0,Y 587.262,Z 578.943,A -85,B 0,C 180,E1 -1353.259,E2 -1353.259} C_VEL
LIN {X 0,Y 587.31,Z 571.251,A -85,B 0,C 180,E1 -1354.289,E2 -1354.289} C_VEL
LIN {X 0,Y 587.401,Z 562.033,A -85,B 0,C 180,E1 -1355.32,E2 -1355.32} C_VEL
LIN {X 0,Y 587.503,Z 551.675,A -85,B 0,C 180,E1 -1356.281,E2 -1356.281} C_VEL
LIN {X 0,Y 587.595,Z 540.688,A -85,B 0,C 180,E1 -1357.128,E2 -1357.128} C_VEL
LIN {X 0,Y 587.647,Z 528.395,A -85,B 0,C 180,E1 -1357.905,E2 -1357.905} C_VEL
LIN {X 0,Y 587.775,Z 514.622,A -85,B 0,C 180,E1 -1358.596,E2 -1358.596} C_VEL
LIN {X 0,Y 587.88,Z 501.104,A -85,B 0,C 180,E1 -1359.114,E2 -1359.114} C_VEL
LIN {X 0,Y 587.957,Z 487.086,A -85,B 0,C 180,E1 -1359.503,E2 -1359.503} C_VEL
LIN {X 0,Y 588.017,Z 472.237,A -85,B 0,C 180,E1 -1359.763,E2 -1359.763} C_VEL
LIN {X 0,Y 588.079,Z 345.86,A -85,B 0,C 180,E1 -1361.33,E2 -1361.33} C_VEL
LIN {X 0,Y 587.486,Z 342.614,A -85,B 0,C 180,E1 -1361.407,E2 -1361.407} C_VEL
LIN {X 0,Y 587.578,Z 325.156,A -85,B 0,C 180,E1 -1364.015,E2 -1364.015} C_VEL
LIN {X 0,Y 587.638,Z 313.44,A -85,B 0,C 180,E1 -1365.788,E2 -1365.788} C_VEL
LIN {X 0,Y 587.326,Z 310.95,A -85,B 0,C 180,E1 -1366.198,E2 -1366.198} C_VEL
LIN {X 0,Y 587.313,Z 310.956,A -85,B 0,C 180,E1 -1369.03,E2 -1369.03} C_VEL
LIN {X 0,Y 587.276,Z 310.951,A -85,B 0,C 180,E1 -1371.776,E2 -1371.776} C_VEL
LIN {X 0,Y 587.285,Z 310.955,A -85,B 0,C 180,E1 -1374.564,E2 -1374.564} C_VEL
LIN {X 0,Y 587.295,Z 310.956,A -85,B 0,C 180,E1 -1377.048,E2 -1377.048} C_VEL
LIN {X 0,Y 587.284,Z 310.952,A -85,B 0,C 180,E1 -1379.383,E2 -1379.383} C_VEL
LIN {X 0,Y 587.297,Z 310.948,A -85,B 0,C 180,E1 -1381.827,E2 -1381.827} C_VEL
LIN {X 0,Y 587.298,Z 310.953,A -85,B 0,C 180,E1 -1385.058,E2 -1385.058} C_VEL
LIN {X 0,Y 587.278,Z 310.95,A -85,B 0,C 180,E1 -1387.83,E2 -1387.83} C_VEL
LIN {X 0,Y 587.297,Z 310.951,A -85,B 0,C 180,E1 -1390.256,E2 -1390.256} C_VEL
LIN {X 0,Y 587.275,Z 310.954,A -85,B 0,C 180,E1 -1393.113,E2 -1393.113} C_VEL
LIN {X 0,Y 587.289,Z 310.95,A -85,B 0,C 180,E1 -1396.046,E2 -1396.046} C_VEL
LIN {X 0,Y 587.294,Z 310.953,A -85,B 0,C 180,E1 -1398.93,E2 -1398.93} C_VEL
LIN {X 0,Y 587.272,Z 310.951,A -85,B 0,C 180,E1 -1401.516,E2 -1401.516} C_VEL
LIN {X 0,Y 587.273,Z 310.954,A -85,B 0,C 180,E1 -1404.098,E2 -1404.098} C_VEL
LIN {X 0,Y 587.316,Z 310.954,A -85,B 0,C 180,E1 -1406.602,E2 -1406.602} C_VEL
LIN {X 0,Y 587.306,Z 310.949,A -85,B 0,C 180,E1 -1409.032,E2 -1409.032} C_VEL
LIN {X 0,Y 587.273,Z 310.95,A -85,B 0,C 180,E1 -1411.4,E2 -1411.4} C_VEL
LIN {X 0,Y 587.307,Z 310.948,A -85,B 0,C 180,E1 -1413.83,E2 -1413.83} C_VEL
LIN {X 0,Y 587.291,Z 310.952,A -85,B 0,C 180,E1 -1416.74,E2 -1416.74} C_VEL
LIN {X 0,Y 587.305,Z 310.946,A -85,B 0,C 180,E1 -1419.694,E2 -1419.694} C_VEL
LIN {X 0,Y 587.28,Z 310.952,A -85,B 0,C 180,E1 -1421.872,E2 -1421.872} C_VEL
LIN {X 0,Y 587.306,Z 310.95,A -85,B 0,C 180,E1 -1424.736,E2 -1424.736} C_VEL
LIN {X 0,Y 587.281,Z 310.95,A -85,B 0,C 180,E1 -1426.857,E2 -1426.857} C_VEL
LIN {X 0,Y 587.326,Z 310.944,A -85,B 0,C 180,E1 -1429.66,E2 -1429.66} C_VEL
LIN {X 0,Y 587.349,Z 310.947,A -85,B 0,C 180,E1 -1432.436,E2 -1432.436} C_VEL
LIN {X 0,Y 587.335,Z 310.943,A -85,B 0,C 180,E1 -1435.195,E2 -1435.195} C_VEL
LIN {X 0,Y 587.365,Z 310.946,A -85,B 0,C 180,E1 -1437.943,E2 -1437.943} C_VEL
LIN {X 0,Y 587.387,Z 310.938,A -85,B 0,C 180,E1 -1440.685,E2 -1440.685} C_VEL
LIN {X 0,Y 587.363,Z 310.941,A -85,B 0,C 180,E1 -1442.743,E2 -1442.743} C_VEL
LIN {X 0,Y 587.336,Z 310.945,A -85,B 0,C 180,E1 -1445.493,E2 -1445.493} C_VEL
LIN {X 0,Y 587.343,Z 310.948,A -85,B 0,C 180,E1 -1448.255,E2 -1448.255} C_VEL
LIN {X 0,Y 587.354,Z 310.941,A -85,B 0,C 180,E1 -1451.133,E2 -1451.133} C_VEL
LIN {X 0,Y 587.369,Z 310.943,A -85,B 0,C 180,E1 -1454.26,E2 -1454.26} C_VEL
LIN {X 0,Y 587.312,Z 310.949,A -85,B 0,C 180,E1 -1457.407,E2 -1457.407} C_VEL
LIN {X 0,Y 587.311,Z 310.952,A -85,B 0,C 180,E1 -1459.576,E2 -1459.576} C_VEL
LIN {X 0,Y 587.319,Z 310.955,A -85,B 0,C 180,E1 -1461.774,E2 -1461.774} C_VEL
LIN {X 0,Y 587.35,Z 310.941,A -85,B 0,C 180,E1 -1464.758,E2 -1464.758} C_VEL
LIN {X 0,Y 587.313,Z 310.947,A -85,B 0,C 180,E1 -1467.047,E2 -1467.047} C_VEL
LIN {X 0,Y 587.345,Z 310.946,A -85,B 0,C 180,E1 -1469.38,E2 -1469.38} C_VEL
LIN {X 0,Y 587.346,Z 310.95,A -85,B 0,C 180,E1 -1471.835,E2 -1471.835} C_VEL
LIN {X 0,Y 587.345,Z 310.943,A -85,B 0,C 180,E1 -1474.347,E2 -1474.347} C_VEL
LIN {X 0,Y 587.321,Z 310.945,A -85,B 0,C 180,E1 -1476.749,E2 -1476.749} C_VEL
LIN {X 0,Y 587.329,Z 310.95,A -85,B 0,C 180,E1 -1479.361,E2 -1479.361} C_VEL
LIN {X 0,Y 587.338,Z 310.945,A -85,B 0,C 180,E1 -1482.108,E2 -1482.108} C_VEL
LIN {X 0,Y 587.291,Z 310.952,A -85,B 0,C 180,E1 -1485.086,E2 -1485.086} C_VEL
LIN {X 0,Y 587.324,Z 310.948,A -85,B 0,C 180,E1 -1487.925,E2 -1487.925} C_VEL
LIN {X 0,Y 587.332,Z 310.944,A -85,B 0,C 180,E1 -1490.639,E2 -1490.639} C_VEL
LIN {X 0,Y 587.355,Z 310.949,A -85,B 0,C 180,E1 -1493.292,E2 -1493.292} C_VEL
LIN {X 0,Y 587.364,Z 310.944,A -85,B 0,C 180,E1 -1495.78,E2 -1495.78} C_VEL
LIN {X 0,Y 587.342,Z 310.943,A -85,B 0,C 180,E1 -1498.231,E2 -1498.231} C_VEL
LIN {X 0,Y 587.352,Z 310.945,A -85,B 0,C 180,E1 -1500.866,E2 -1500.866} C_VEL
LIN {X 0,Y 587.36,Z 310.944,A -85,B 0,C 180,E1 -1503.819,E2 -1503.819} C_VEL
LIN {X 0,Y 587.379,Z 311.084,A -85,B 0,C 180,E1 -1505.809,E2 -1505.809} C_VEL
LIN {X 0,Y 588,Z 315.314,A -85,B 0,C 180,E1 -1506.396,E2 -1506.396} C_VEL
LIN {X 0,Y 587.841,Z 335.098,A -85,B 0,C 180,E1 -1508.981,E2 -1508.981} C_VEL
LIN {X 0,Y 587.701,Z 357.707,A -85,B 0,C 180,E1 -1511.885,E2 -1511.885} C_VEL
LIN {X 0,Y 587.583,Z 371.572,A -85,B 0,C 180,E1 -1513.642,E2 -1513.642} C_VEL
LIN {X 0,Y 588.227,Z 375.607,A -85,B 0,C 180,E1 -1513.716,E2 -1513.716} C_VEL
LIN {X 0,Y 588.013,Z 509.88,A -85,B 0,C 180,E1 -1515.397,E2 -1515.397} C_VEL
LIN {X 0,Y 587.936,Z 524.08,A -85,B 0,C 180,E1 -1515.718,E2 -1515.718} C_VEL
LIN {X 0,Y 587.824,Z 537.711,A -85,B 0,C 180,E1 -1516.165,E2 -1516.165} C_VEL
LIN {X 0,Y 587.727,Z 551.637,A -85,B 0,C 180,E1 -1516.78,E2 -1516.78} C_VEL
LIN {X 0,Y 587.605,Z 564.096,A -85,B 0,C 180,E1 -1517.48,E2 -1517.48} C_VEL
LIN {X 0,Y 587.513,Z 576.638,A -85,B 0,C 180,E1 -1518.354,E2 -1518.354} C_VEL
LIN {X 0,Y 587.444,Z 587.835,A -85,B 0,C 180,E1 -1519.313,E2 -1519.313} C_VEL
LIN {X 0,Y 587.319,Z 597.85,A -85,B 0,C 180,E1 -1520.356,E2 -1520.356} C_VEL
LIN {X 0,Y 587.277,Z 606.17,A -85,B 0,C 180,E1 -1521.397,E2 -1521.397} C_VEL
LIN {X 0,Y 587.244,Z 614.126,A -85,B 0,C 180,E1 -1522.608,E2 -1522.608} C_VEL
LIN {X 0,Y 587.203,Z 620.527,A -85,B 0,C 180,E1 -1523.816,E2 -1523.816} C_VEL
LIN {X 0,Y 587.16,Z 624.961,A -85,B 0,C 180,E1 -1524.85,E2 -1524.85} C_VEL
LIN {X 0,Y 587.179,Z 628.442,A -85,B 0,C 180,E1 -1525.882,E2 -1525.882} C_VEL
LIN {X 0,Y 587.13,Z 631.831,A -85,B 0,C 180,E1 -1527.256,E2 -1527.256} C_VEL
LIN {X 0,Y 587.141,Z 633.832,A -85,B 0,C 180,E1 -1528.628,E2 -1528.628} C_VEL
LIN {X 0,Y 587.135,Z 634.5,A -85,B 0,C 180,E1 -1530,E2 -1530} C_VEL
LIN {X 0,Y 587.141,Z 633.832,A -85,B 0,C 180,E1 -1531.372,E2 -1531.372} C_VEL
LIN {X 0,Y 587.13,Z 631.832,A -85,B 0,C 180,E1 -1532.744,E2 -1532.744} C_VEL
LIN {X 0,Y 587.179,Z 628.443,A -85,B 0,C 180,E1 -1534.118,E2 -1534.118} C_VEL
LIN {X 0,Y 587.199,Z 623.567,A -85,B 0,C 180,E1 -1535.495,E2 -1535.495} C_VEL
LIN {X 0,Y 587.209,Z 617.052,A -85,B 0,C 180,E1 -1536.874,E2 -1536.874} C_VEL
LIN {X 0,Y 587.268,Z 609.799,A -85,B 0,C 180,E1 -1538.084,E2 -1538.084} C_VEL
LIN {X 0,Y 587.321,Z 600.822,A -85,B 0,C 180,E1 -1539.297,E2 -1539.297} C_VEL
LIN {X 0,Y 587.372,Z 591.39,A -85,B 0,C 180,E1 -1540.339,E2 -1540.339} C_VEL
LIN {X 0,Y 587.475,Z 581.026,A -85,B 0,C 180,E1 -1541.29,E2 -1541.29} C_VEL
LIN {X 0,Y 587.575,Z 569.428,A -85,B 0,C 180,E1 -1542.17,E2 -1542.17} C_VEL
LIN {X 0,Y 587.668,Z 556.646,A -85,B 0,C 180,E1 -1542.958,E2 -1542.958} C_VEL
LIN {X 0,Y 587.78,Z 544.156,A -85,B 0,C 180,E1 -1543.571,E2 -1543.571} C_VEL
LIN {X 0,Y 587.889,Z 530.602,A -85,B 0,C 180,E1 -1544.086,E2 -1544.086} C_VEL
LIN {X 0,Y 587.947,Z 516.952,A -85,B 0,C 180,E1 -1544.462,E2 -1544.462} C_VEL
LIN {X 0,Y 588.011,Z 502.591,A -85,B 0,C 180,E1 -1544.713,E2 -1544.713} C_VEL
LIN {X 0,Y 588.058,Z 374.261,A -85,B 0,C 180,E1 -1546.306,E2 -1546.306} C_VEL
LIN {X 0,Y 587.583,Z 371.484,A -85,B 0,C 180,E1 -1546.369,E2 -1546.369} C_VEL
LIN {X 0,Y 587.724,Z 349.635,A -85,B 0,C 180,E1 -1549.147,E2 -1549.147} C_VEL
LIN {X 0,Y 587.884,Z 329.445,A -85,B 0,C 180,E1 -1551.753,E2 -1551.753} C_VEL
LIN {X 0,Y 587.915,Z 313.901,A -85,B 0,C 180,E1 -1553.794,E2 -1553.794} C_VEL
LIN {X 0,Y 587.368,Z 310.947,A -85,B 0,C 180,E1 -1554.213,E2 -1554.213} C_VEL
LIN {X 0,Y 587.329,Z 310.949,A -85,B 0,C 180,E1 -1557.046,E2 -1557.046} C_VEL
LIN {X 0,Y 587.35,Z 310.942,A -85,B 0,C 180,E1 -1559.38,E2 -1559.38} C_VEL
LIN {X 0,Y 587.345,Z 310.943,A -85,B 0,C 180,E1 -1561.836,E2 -1561.836} C_VEL
LIN {X 0,Y 587.35,Z 310.947,A -85,B 0,C 180,E1 -1564.348,E2 -1564.348} C_VEL
LIN {X 0,Y 587.344,Z 310.942,A -85,B 0,C 180,E1 -1567.608,E2 -1567.608} C_VEL
LIN {X 0,Y 587.314,Z 310.952,A -85,B 0,C 180,E1 -1570.255,E2 -1570.255} C_VEL
LIN {X 0,Y 587.314,Z 310.947,A -85,B 0,C 180,E1 -1573.118,E2 -1573.118} C_VEL
LIN {X 0,Y 587.315,Z 310.949,A -85,B 0,C 180,E1 -1576.049,E2 -1576.049} C_VEL
LIN {X 0,Y 587.334,Z 310.946,A -85,B 0,C 180,E1 -1578.926,E2 -1578.926} C_VEL
LIN {X 0,Y 587.322,Z 310.945,A -85,B 0,C 180,E1 -1581.52,E2 -1581.52} C_VEL
LIN {X 0,Y 587.298,Z 310.956,A -85,B 0,C 180,E1 -1584.463,E2 -1584.463} C_VEL
LIN {X 0,Y 587.34,Z 310.944,A -85,B 0,C 180,E1 -1586.889,E2 -1586.889} C_VEL
LIN {X 0,Y 587.334,Z 310.947,A -85,B 0,C 180,E1 -1589.83,E2 -1589.83} C_VEL
LIN {X 0,Y 587.304,Z 310.956,A -85,B 0,C 180,E1 -1592.317,E2 -1592.317} C_VEL
LIN {X 0,Y 587.356,Z 310.941,A -85,B 0,C 180,E1 -1595.42,E2 -1595.42} C_VEL
LIN {X 0,Y 587.319,Z 310.954,A -85,B 0,C 180,E1 -1598.226,E2 -1598.226} C_VEL
LIN {X 0,Y 587.345,Z 310.942,A -85,B 0,C 180,E1 -1601.151,E2 -1601.151} C_VEL
LIN {X 0,Y 587.316,Z 310.955,A -85,B 0,C 180,E1 -1604.025,E2 -1604.025} C_VEL
LIN {X 0,Y 587.356,Z 310.949,A -85,B 0,C 180,E1 -1606.154,E2 -1606.154} C_VEL
LIN {X 0,Y 587.342,Z 310.942,A -85,B 0,C 180,E1 -1608.963,E2 -1608.963} C_VEL
LIN {X 0,Y 587.343,Z 310.948,A -85,B 0,C 180,E1 -1611.745,E2 -1611.745} C_VEL
LIN {X 0,Y 587.335,Z 310.945,A -85,B 0,C 180,E1 -1614.507,E2 -1614.507} C_VEL
LIN {X 0,Y 587.364,Z 310.94,A -85,B 0,C 180,E1 -1617.257,E2 -1617.257} C_VEL
LIN {X 0,Y 587.38,Z 310.946,A -85,B 0,C 180,E1 -1620,E2 -1620} C_VEL
LIN {X 0,Y 587.347,Z 310.941,A -85,B 0,C 180,E1 -1622.744,E2 -1622.744} C_VEL
LIN {X 0,Y 587.349,Z 310.946,A -85,B 0,C 180,E1 -1625.493,E2 -1625.493} C_VEL
LIN {X 0,Y 587.322,Z 310.948,A -85,B 0,C 180,E1 -1628.256,E2 -1628.256} C_VEL
LIN {X 0,Y 587.336,Z 310.944,A -85,B 0,C 180,E1 -1631.124,E2 -1631.124} C_VEL
LIN {X 0,Y 587.323,Z 310.947,A -85,B 0,C 180,E1 -1634.242,E2 -1634.242} C_VEL
LIN {X 0,Y 587.281,Z 310.949,A -85,B 0,C 180,E1 -1636.79,E2 -1636.79} C_VEL
LIN {X 0,Y 587.281,Z 310.952,A -85,B 0,C 180,E1 -1638.266,E2 -1638.266} C_VEL
LIN {X 0,Y 586.628,Z 311.033,A -85,B 0,C 180,E1 -1638.838,E2 -1638.838} C_VEL
LIN {X 0,Y 583.773,Z 311.394,A -85,B 0,C 180,E1 -1639.766,E2 -1639.766} C_VEL
LIN {X 0,Y 581.363,Z 311.69,A -85,B 0,C 180,E1 -1640.513,E2 -1640.513} C_VEL
LIN {X 0,Y 580.344,Z 311.816,A -85,B 0,C 180,E1 -1641.09,E2 -1641.09} C_VEL
LIN {X 0,Y 580.27,Z 311.827,A -85,B 0,C 180,E1 -1641.285,E2 -1641.285} C_VEL
LIN {X 0,Y 580.25,Z 311.826,A -85,B 0,C 180,E1 -1644.319,E2 -1644.319} C_VEL
LIN {X 0,Y 580.243,Z 311.827,A -85,B 0,C 180,E1 -1646.625,E2 -1646.625} C_VEL
LIN {X 0,Y 580.252,Z 311.831,A -85,B 0,C 180,E1 -1649.3,E2 -1649.3} C_VEL
LIN {X 0,Y 580.279,Z 311.823,A -85,B 0,C 180,E1 -1652.202,E2 -1652.202} C_VEL
LIN {X 0,Y 580.272,Z 311.824,A -85,B 0,C 180,E1 -1654.698,E2 -1654.698} C_VEL
LIN {X 0,Y 580.268,Z 311.829,A -85,B 0,C 180,E1 -1657.271,E2 -1657.271} C_VEL
LIN {X 0,Y 580.241,Z 311.827,A -85,B 0,C 180,E1 -1660.264,E2 -1660.264} C_VEL
LIN {X 0,Y 580.244,Z 311.828,A -85,B 0,C 180,E1 -1662.71,E2 -1662.71} C_VEL
LIN {X 0,Y 580.23,Z 311.833,A -85,B 0,C 180,E1 -1665.614,E2 -1665.614} C_VEL
LIN {X 0,Y 580.209,Z 311.831,A -85,B 0,C 180,E1 -1668.225,E2 -1668.225} C_VEL
LIN {X 0,Y 580.237,Z 311.833,A -85,B 0,C 180,E1 -1670.961,E2 -1670.961} C_VEL
LIN {X 0,Y 580.23,Z 311.833,A -85,B 0,C 180,E1 -1673.593,E2 -1673.593} C_VEL
LIN {X 0,Y 580.255,Z 311.826,A -85,B 0,C 180,E1 -1676.141,E2 -1676.141} C_VEL
LIN {X 0,Y 580.24,Z 311.83,A -85,B 0,C 180,E1 -1678.612,E2 -1678.612} C_VEL
LIN {X 0,Y 580.248,Z 311.836,A -85,B 0,C 180,E1 -1681.021,E2 -1681.021} C_VEL
LIN {X 0,Y 580.288,Z 311.984,A -85,B 0,C 180,E1 -1683.801,E2 -1683.801} C_VEL
LIN {X 0,Y 580.729,Z 316.768,A -85,B 0,C 180,E1 -1684.556,E2 -1684.556} C_VEL
LIN {X 0,Y 580.57,Z 335.418,A -85,B 0,C 180,E1 -1687.397,E2 -1687.397} C_VEL
LIN {X 0,Y 580.498,Z 342.674,A -85,B 0,C 180,E1 -1688.49,E2 -1688.49} C_VEL
LIN {X 0,Y 581.378,Z 348.73,A -85,B 0,C 180,E1 -1688.603,E2 -1688.603} C_VEL
LIN {X 0,Y 581.125,Z 479.683,A -85,B 0,C 180,E1 -1690.261,E2 -1690.261} C_VEL
LIN {X 0,Y 581.04,Z 494.328,A -85,B 0,C 180,E1 -1690.597,E2 -1690.597} C_VEL
LIN {X 0,Y 580.943,Z 508.449,A -85,B 0,C 180,E1 -1691.073,E2 -1691.073} C_VEL
LIN {X 0,Y 580.808,Z 521.608,A -85,B 0,C 180,E1 -1691.663,E2 -1691.663} C_VEL
LIN {X 0,Y 580.652,Z 534.324,A -85,B 0,C 180,E1 -1692.387,E2 -1692.387} C_VEL
LIN {X 0,Y 580.535,Z 545.888,A -85,B 0,C 180,E1 -1693.2,E2 -1693.2} C_VEL
LIN {X 0,Y 580.426,Z 557.454,A -85,B 0,C 180,E1 -1694.19,E2 -1694.19} C_VEL
LIN {X 0,Y 580.313,Z 567.707,A -85,B 0,C 180,E1 -1695.266,E2 -1695.266} C_VEL
LIN {X 0,Y 580.227,Z 576.181,A -85,B 0,C 180,E1 -1696.338,E2 -1696.338} C_VEL
LIN {X 0,Y 580.153,Z 584.246,A -85,B 0,C 180,E1 -1697.583,E2 -1697.583} C_VEL
LIN {X 0,Y 580.081,Z 591.16,A -85,B 0,C 180,E1 -1698.922,E2 -1698.922} C_VEL
LIN {X 0,Y 580.084,Z 596.393,A -85,B 0,C 180,E1 -1700.234,E2 -1700.234} C_VEL
LIN {X 0,Y 580.069,Z 600.491,A -85,B 0,C 180,E1 -1701.64,E2 -1701.64} C_VEL
LIN {X 0,Y 580.061,Z 603.124,A -85,B 0,C 180,E1 -1703.041,E2 -1703.041} C_VEL
LIN {X 0,Y 580.086,Z 604.369,A -85,B 0,C 180,E1 -1704.438,E2 -1704.438} C_VEL
LIN {X 0,Y 580.085,Z 604.271,A -85,B 0,C 180,E1 -1705.831,E2 -1705.831} C_VEL
LIN {X 0,Y 580.035,Z 602.852,A -85,B 0,C 180,E1 -1707.222,E2 -1707.222} C_VEL
LIN {X 0,Y 580.049,Z 600.078,A -85,B 0,C 180,E1 -1708.611,E2 -1708.611} C_VEL
LIN {X 0,Y 580.07,Z 595.881,A -85,B 0,C 180,E1 -1710,E2 -1710} C_VEL
LIN {X 0,Y 580.082,Z 590.141,A -85,B 0,C 180,E1 -1711.388,E2 -1711.388} C_VEL
LIN {X 0,Y 580.209,Z 583.684,A -85,B 0,C 180,E1 -1712.603,E2 -1712.603} C_VEL
LIN {X 0,Y 580.26,Z 575.702,A -85,B 0,C 180,E1 -1713.82,E2 -1713.82} C_VEL
LIN {X 0,Y 580.352,Z 567.371,A -85,B 0,C 180,E1 -1714.863,E2 -1714.863} C_VEL
LIN {X 0,Y 580.421,Z 557.372,A -85,B 0,C 180,E1 -1715.907,E2 -1715.907} C_VEL
LIN {X 0,Y 580.517,Z 546.94,A -85,B 0,C 180,E1 -1716.81,E2 -1716.81} C_VEL
LIN {X 0,Y 580.656,Z 535.154,A -85,B 0,C 180,E1 -1717.651,E2 -1717.651} C_VEL
LIN {X 0,Y 580.784,Z 523.148,A -85,B 0,C 180,E1 -1718.35,E2 -1718.35} C_VEL
LIN {X 0,Y 580.932,Z 509.882,A -85,B 0,C 180,E1 -1718.961,E2 -1718.961} C_VEL
LIN {X 0,Y 581.059,Z 496.058,A -85,B 0,C 180,E1 -1719.442,E2 -1719.442} C_VEL
LIN {X 0,Y 581.132,Z 481.553,A -85,B 0,C 180,E1 -1719.792,E2 -1719.792} C_VEL
LIN {X 0,Y 581.178,Z 457.817,A -85,B 0,C 180,E1 -1720.121,E2 -1720.121} C_VEL
LIN {X 0,Y 581.372,Z 347.428,A -85,B 0,C 180,E1 -1721.504,E2 -1721.504} C_VEL
LIN {X 0,Y 580.485,Z 342.747,A -85,B 0,C 180,E1 -1721.59,E2 -1721.59} C_VEL
LIN {X 0,Y 580.598,Z 326.742,A -85,B 0,C 180,E1 -1724.01,E2 -1724.01} C_VEL
LIN {X 0,Y 580.698,Z 315.035,A -85,B 0,C 180,E1 -1725.802,E2 -1725.802} C_VEL
LIN {X 0,Y 580.282,Z 311.829,A -85,B 0,C 180,E1 -1726.333,E2 -1726.333} C_VEL
LIN {X 0,Y 580.27,Z 311.832,A -85,B 0,C 180,E1 -1729.141,E2 -1729.141} C_VEL
LIN {X 0,Y 580.23,Z 311.829,A -85,B 0,C 180,E1 -1732.054,E2 -1732.054} C_VEL
LIN {X 0,Y 580.239,Z 311.835,A -85,B 0,C 180,E1 -1734.711,E2 -1734.711} C_VEL
LIN {X 0,Y 580.238,Z 311.83,A -85,B 0,C 180,E1 -1737.404,E2 -1737.404} C_VEL
LIN {X 0,Y 580.23,Z 311.828,A -85,B 0,C 180,E1 -1739.776,E2 -1739.776} C_VEL
LIN {X 0,Y 580.272,Z 311.825,A -85,B 0,C 180,E1 -1742.202,E2 -1742.202} C_VEL
LIN {X 0,Y 580.265,Z 311.833,A -85,B 0,C 180,E1 -1744.698,E2 -1744.698} C_VEL
LIN {X 0,Y 580.26,Z 311.827,A -85,B 0,C 180,E1 -1747.272,E2 -1747.272} C_VEL
LIN {X 0,Y 580.278,Z 311.826,A -85,B 0,C 180,E1 -1750.268,E2 -1750.268} C_VEL
LIN {X 0,Y 580.243,Z 311.837,A -85,B 0,C 180,E1 -1752.71,E2 -1752.71} C_VEL
LIN {X 0,Y 580.236,Z 311.827,A -85,B 0,C 180,E1 -1755.613,E2 -1755.613} C_VEL
LIN {X 0,Y 580.238,Z 311.831,A -85,B 0,C 180,E1 -1758.227,E2 -1758.227} C_VEL
LIN {X 0,Y 580.24,Z 311.831,A -85,B 0,C 180,E1 -1760.962,E2 -1760.962} C_VEL
LIN {X 0,Y 580.239,Z 311.827,A -85,B 0,C 180,E1 -1763.594,E2 -1763.594} C_VEL
LIN {X 0,Y 580.27,Z 311.827,A -85,B 0,C 180,E1 -1766.142,E2 -1766.142} C_VEL
LIN {X 0,Y 580.263,Z 311.832,A -85,B 0,C 180,E1 -1768.613,E2 -1768.613} C_VEL
LIN {X 0,Y 580.249,Z 311.827,A -85,B 0,C 180,E1 -1771.021,E2 -1771.021} C_VEL
LIN {X 0,Y 580.262,Z 311.824,A -85,B 0,C 180,E1 -1773.673,E2 -1773.673} C_VEL
LIN {X 0,Y 580.246,Z 311.835,A -85,B 0,C 180,E1 -1776.44,E2 -1776.44} C_VEL
LIN {X 0,Y 580.254,Z 311.823,A -85,B 0,C 180,E1 -1779.436,E2 -1779.436} C_VEL
LIN {X 0,Y 580.24,Z 311.827,A -85,B 0,C 180,E1 -1781.644,E2 -1781.644} C_VEL
LIN {X 0,Y 580.273,Z 311.829,A -85,B 0,C 180,E1 -1784.546,E2 -1784.546} C_VEL
LIN {X 0,Y 580.242,Z 311.829,A -85,B 0,C 180,E1 -1786.695,E2 -1786.695} C_VEL
LIN {X 0,Y 580.311,Z 311.816,A -85,B 0,C 180,E1 -1788.827,E2 -1788.827} C_VEL
LIN {X 0,Y 580.303,Z 311.82,A -85,B 0,C 180,E1 -1791.643,E2 -1791.643} C_VEL
LIN {X 0,Y 580.315,Z 311.823,A -85,B 0,C 180,E1 -1794.44,E2 -1794.44} C_VEL
LIN {X 0,Y 580.318,Z 311.817,A -85,B 0,C 180,E1 -1797.223,E2 -1797.223} C_VEL
LIN {X 0,Y 580.349,Z 311.822,A -85,B 0,C 180,E1 -1800,E2 -1800} C_VEL
LIN {X 0,Y 580.328,Z 311.817,A -85,B 0,C 180,E1 -1802.776,E2 -1802.776} C_VEL
LIN {X 0,Y 580.305,Z 311.821,A -85,B 0,C 180,E1 -1805.56,E2 -1805.56} C_VEL
LIN {X 0,Y 580.311,Z 311.822,A -85,B 0,C 180,E1 -1808.356,E2 -1808.356} C_VEL
LIN {X 0,Y 580.305,Z 311.819,A -85,B 0,C 180,E1 -1811.191,E2 -1811.191} C_VEL
LIN {X 0,Y 580.326,Z 311.825,A -85,B 0,C 180,E1 -1814.017,E2 -1814.017} C_VEL
LIN {X 0,Y 580.317,Z 311.817,A -85,B 0,C 180,E1 -1816.914,E2 -1816.914} C_VEL
LIN {X 0,Y 580.286,Z 311.831,A -85,B 0,C 180,E1 -1819.823,E2 -1819.823} C_VEL
LIN {X 0,Y 580.271,Z 311.829,A -85,B 0,C 180,E1 -1822.053,E2 -1822.053} C_VEL
LIN {X 0,Y 580.306,Z 311.82,A -85,B 0,C 180,E1 -1825.08,E2 -1825.08} C_VEL
LIN {X 0,Y 580.282,Z 311.825,A -85,B 0,C 180,E1 -1828.186,E2 -1828.186} C_VEL
LIN {X 0,Y 580.284,Z 311.822,A -85,B 0,C 180,E1 -1830.694,E2 -1830.694} C_VEL
LIN {X 0,Y 580.304,Z 311.823,A -85,B 0,C 180,E1 -1833.316,E2 -1833.316} C_VEL
LIN {X 0,Y 580.262,Z 311.833,A -85,B 0,C 180,E1 -1835.758,E2 -1835.758} C_VEL
LIN {X 0,Y 580.287,Z 311.823,A -85,B 0,C 180,E1 -1838.146,E2 -1838.146} C_VEL
LIN {X 0,Y 580.297,Z 311.821,A -85,B 0,C 180,E1 -1840.844,E2 -1840.844} C_VEL
LIN {X 0,Y 580.274,Z 311.831,A -85,B 0,C 180,E1 -1843.658,E2 -1843.658} C_VEL
LIN {X 0,Y 580.274,Z 311.823,A -85,B 0,C 180,E1 -1846.61,E2 -1846.61} C_VEL
LIN {X 0,Y 580.297,Z 311.825,A -85,B 0,C 180,E1 -1849.156,E2 -1849.156} C_VEL
LIN {X 0,Y 580.291,Z 311.824,A -85,B 0,C 180,E1 -1851.927,E2 -1851.927} C_VEL
LIN {X 0,Y 580.287,Z 311.822,A -85,B 0,C 180,E1 -1854.455,E2 -1854.455} C_VEL
LIN {X 0,Y 580.291,Z 311.825,A -85,B 0,C 180,E1 -1856.975,E2 -1856.975} C_VEL
LIN {X 0,Y 580.296,Z 311.83,A -85,B 0,C 180,E1 -1859.425,E2 -1859.425} C_VEL
LIN {X 0,Y 580.294,Z 311.822,A -85,B 0,C 180,E1 -1862.142,E2 -1862.142} C_VEL
LIN {X 0,Y 580.323,Z 311.826,A -85,B 0,C 180,E1 -1865.27,E2 -1865.27} C_VEL
LIN {X 0,Y 580.373,Z 312.02,A -85,B 0,C 180,E1 -1865.624,E2 -1865.624} C_VEL
LIN {X 0,Y 581.126,Z 316.728,A -85,B 0,C 180,E1 -1866.289,E2 -1866.289} C_VEL
LIN {X 0,Y 580.937,Z 336.511,A -85,B 0,C 180,E1 -1868.905,E2 -1868.905} C_VEL
LIN {X 0,Y 580.744,Z 359.12,A -85,B 0,C 180,E1 -1871.843,E2 -1871.843} C_VEL
LIN {X 0,Y 580.598,Z 371.617,A -85,B 0,C 180,E1 -1873.445,E2 -1873.445} C_VEL
LIN {X 0,Y 581.398,Z 377.395,A -85,B 0,C 180,E1 -1873.542,E2 -1873.542} C_VEL
LIN {X 0,Y 581.145,Z 509.88,A -85,B 0,C 180,E1 -1875.221,E2 -1875.221} C_VEL
LIN {X 0,Y 581.06,Z 524.229,A -85,B 0,C 180,E1 -1875.55,E2 -1875.55} C_VEL
LIN {X 0,Y 580.919,Z 537.709,A -85,B 0,C 180,E1 -1875.998,E2 -1875.998} C_VEL
LIN {X 0,Y 580.787,Z 551.639,A -85,B 0,C 180,E1 -1876.619,E2 -1876.619} C_VEL
LIN {X 0,Y 580.656,Z 564.098,A -85,B 0,C 180,E1 -1877.328,E2 -1877.328} C_VEL
LIN {X 0,Y 580.526,Z 576.64,A -85,B 0,C 180,E1 -1878.212,E2 -1878.212} C_VEL
LIN {X 0,Y 580.441,Z 587.905,A -85,B 0,C 180,E1 -1879.19,E2 -1879.19} C_VEL
LIN {X 0,Y 580.275,Z 597.851,A -85,B 0,C 180,E1 -1880.238,E2 -1880.238} C_VEL
LIN {X 0,Y 580.241,Z 606.171,A -85,B 0,C 180,E1 -1881.292,E2 -1881.292} C_VEL
LIN {X 0,Y 580.165,Z 614.126,A -85,B 0,C 180,E1 -1882.517,E2 -1882.517} C_VEL
LIN {X 0,Y 580.102,Z 620.527,A -85,B 0,C 180,E1 -1883.74,E2 -1883.74} C_VEL
LIN {X 0,Y 580.078,Z 624.961,A -85,B 0,C 180,E1 -1884.786,E2 -1884.786} C_VEL
LIN {X 0,Y 580.102,Z 628.443,A -85,B 0,C 180,E1 -1885.831,E2 -1885.831} C_VEL
LIN {X 0,Y 580.041,Z 631.832,A -85,B 0,C 180,E1 -1887.222,E2 -1887.222} C_VEL
LIN {X 0,Y 580.041,Z 633.832,A -85,B 0,C 180,E1 -1888.611,E2 -1888.611} C_VEL
LIN {X 0,Y 580.036,Z 634.5,A -85,B 0,C 180,E1 -1890,E2 -1890} C_VEL
LIN {X 0,Y 580.041,Z 633.833,A -85,B 0,C 180,E1 -1891.389,E2 -1891.389} C_VEL
LIN {X 0,Y 580.041,Z 631.833,A -85,B 0,C 180,E1 -1892.778,E2 -1892.778} C_VEL
LIN {X 0,Y 580.102,Z 628.444,A -85,B 0,C 180,E1 -1894.169,E2 -1894.169} C_VEL
LIN {X 0,Y 580.128,Z 623.568,A -85,B 0,C 180,E1 -1895.562,E2 -1895.562} C_VEL
LIN {X 0,Y 580.141,Z 617.052,A -85,B 0,C 180,E1 -1896.958,E2 -1896.958} C_VEL
LIN {X 0,Y 580.192,Z 609.799,A -85,B 0,C 180,E1 -1898.183,E2 -1898.183} C_VEL
LIN {X 0,Y 580.284,Z 600.822,A -85,B 0,C 180,E1 -1899.41,E2 -1899.41} C_VEL
LIN {X 0,Y 580.356,Z 591.39,A -85,B 0,C 180,E1 -1900.466,E2 -1900.466} C_VEL
LIN {X 0,Y 580.476,Z 581.318,A -85,B 0,C 180,E1 -1901.404,E2 -1901.404} C_VEL
LIN {X 0,Y 580.597,Z 569.43,A -85,B 0,C 180,E1 -1902.319,E2 -1902.319} C_VEL
LIN {X 0,Y 580.731,Z 556.644,A -85,B 0,C 180,E1 -1903.115,E2 -1903.115} C_VEL
LIN {X 0,Y 580.86,Z 544.153,A -85,B 0,C 180,E1 -1903.736,E2 -1903.736} C_VEL
LIN {X 0,Y 581.01,Z 531.18,A -85,B 0,C 180,E1 -1904.236,E2 -1904.236} C_VEL
LIN {X 0,Y 581.084,Z 517.163,A -85,B 0,C 180,E1 -1904.631,E2 -1904.631} C_VEL
LIN {X 0,Y 581.159,Z 502.591,A -85,B 0,C 180,E1 -1904.891,E2 -1904.891} C_VEL
LIN {X 0,Y 581.274,Z 375.277,A -85,B 0,C 180,E1 -1906.489,E2 -1906.489} C_VEL
LIN {X 0,Y 580.603,Z 371.484,A -85,B 0,C 180,E1 -1906.572,E2 -1906.572} C_VEL
LIN {X 0,Y 580.803,Z 350.329,A -85,B 0,C 180,E1 -1909.294,E2 -1909.294} C_VEL
LIN {X 0,Y 581.045,Z 328.032,A -85,B 0,C 180,E1 -1912.209,E2 -1912.209} C_VEL
LIN {X 0,Y 581.023,Z 315.314,A -85,B 0,C 180,E1 -1913.905,E2 -1913.905} C_VEL
LIN {X 0,Y 580.342,Z 311.824,A -85,B 0,C 180,E1 -1914.441,E2 -1914.441} C_VEL
LIN {X 0,Y 580.283,Z 311.824,A -85,B 0,C 180,E1 -1917.402,E2 -1917.402} C_VEL
LIN {X 0,Y 580.291,Z 311.821,A -85,B 0,C 180,E1 -1919.773,E2 -1919.773} C_VEL
LIN {X 0,Y 580.3,Z 311.823,A -85,B 0,C 180,E1 -1922.201,E2 -1922.201} C_VEL
LIN {X 0,Y 580.292,Z 311.83,A -85,B 0,C 180,E1 -1924.696,E2 -1924.696} C_VEL
LIN {X 0,Y 580.299,Z 311.821,A -85,B 0,C 180,E1 -1927.269,E2 -1927.269} C_VEL
LIN {X 0,Y 580.293,Z 311.826,A -85,B 0,C 180,E1 -1930.271,E2 -1930.271} C_VEL
LIN {X 0,Y 580.278,Z 311.829,A -85,B 0,C 180,E1 -1932.707,E2 -1932.707} C_VEL
LIN {X 0,Y 580.258,Z 311.825,A -85,B 0,C 180,E1 -1935.611,E2 -1935.611} C_VEL
LIN {X 0,Y 580.283,Z 311.829,A -85,B 0,C 180,E1 -1938.231,E2 -1938.231} C_VEL
LIN {X 0,Y 580.272,Z 311.825,A -85,B 0,C 180,E1 -1940.965,E2 -1940.965} C_VEL
LIN {X 0,Y 580.251,Z 311.826,A -85,B 0,C 180,E1 -1943.595,E2 -1943.595} C_VEL
LIN {X 0,Y 580.315,Z 311.825,A -85,B 0,C 180,E1 -1946.145,E2 -1946.145} C_VEL
LIN {X 0,Y 580.277,Z 311.827,A -85,B 0,C 180,E1 -1948.615,E2 -1948.615} C_VEL
LIN {X 0,Y 580.291,Z 311.821,A -85,B 0,C 180,E1 -1951.024,E2 -1951.024} C_VEL
LIN {X 0,Y 580.268,Z 311.833,A -85,B 0,C 180,E1 -1954.15,E2 -1954.15} C_VEL
LIN {X 0,Y 580.274,Z 311.828,A -85,B 0,C 180,E1 -1956.442,E2 -1956.442} C_VEL
LIN {X 0,Y 580.273,Z 311.824,A -85,B 0,C 180,E1 -1959.437,E2 -1959.437} C_VEL
LIN {X 0,Y 580.263,Z 311.827,A -85,B 0,C 180,E1 -1961.645,E2 -1961.645} C_VEL
LIN {X 0,Y 580.269,Z 311.829,A -85,B 0,C 180,E1 -1963.825,E2 -1963.825} C_VEL
LIN {X 0,Y 580.326,Z 311.825,A -85,B 0,C 180,E1 -1965.983,E2 -1965.983} C_VEL
LIN {X 0,Y 580.311,Z 311.819,A -85,B 0,C 180,E1 -1968.827,E2 -1968.827} C_VEL
LIN {X 0,Y 580.311,Z 311.822,A -85,B 0,C 180,E1 -1971.644,E2 -1971.644} C_VEL
LIN {X 0,Y 580.304,Z 311.822,A -85,B 0,C 180,E1 -1974.44,E2 -1974.44} C_VEL
LIN {X 0,Y 580.328,Z 311.816,A -85,B 0,C 180,E1 -1977.224,E2 -1977.224} C_VEL
LIN {X 0,Y 580.349,Z 311.821,A -85,B 0,C 180,E1 -1980,E2 -1980} C_VEL
LIN {X 0,Y 580.317,Z 311.817,A -85,B 0,C 180,E1 -1982.777,E2 -1982.777} C_VEL
LIN {X 0,Y 580.314,Z 311.824,A -85,B 0,C 180,E1 -1985.56,E2 -1985.56} C_VEL
LIN {X 0,Y 580.294,Z 311.822,A -85,B 0,C 180,E1 -1988.357,E2 -1988.357} C_VEL
LIN {X 0,Y 580.307,Z 311.82,A -85,B 0,C 180,E1 -1991.191,E2 -1991.191} C_VEL
LIN {X 0,Y 580.285,Z 311.823,A -85,B 0,C 180,E1 -1994.324,E2 -1994.324} C_VEL
LIN {X 0,Y 580.231,Z 311.828,A -85,B 0,C 180,E1 -1996.9,E2 -1996.9} C_VEL
LIN {X 0,Y 580.274,Z 311.829,A -85,B 0,C 180,E1 -1999.824,E2 -1999.824} C_VEL
LIN {X 0,Y 580.27,Z 311.827,A -85,B 0,C 180,E1 -2001.285,E2 -2001.285} C_VEL
LIN {X 0,Y 579.618,Z 311.915,A -85,B 0,C 180,E1 -2001.865,E2 -2001.865} C_VEL
LIN {X 0,Y 576.738,Z 312.273,A -85,B 0,C 180,E1 -2002.804,E2 -2002.804} C_VEL
LIN {X 0,Y 574.302,Z 312.577,A -85,B 0,C 180,E1 -2003.56,E2 -2003.56} C_VEL
LIN {X 0,Y 573.272,Z 312.697,A -85,B 0,C 180,E1 -2004.144,E2 -2004.144} C_VEL
LIN {X 0,Y 573.197,Z 312.704,A -85,B 0,C 180,E1 -2004.342,E2 -2004.342} C_VEL
LIN {X 0,Y 573.191,Z 312.707,A -85,B 0,C 180,E1 -2006.979,E2 -2006.979} C_VEL
LIN {X 0,Y 573.202,Z 312.711,A -85,B 0,C 180,E1 -2009.479,E2 -2009.479} C_VEL
LIN {X 0,Y 573.232,Z 312.7,A -85,B 0,C 180,E1 -2012.224,E2 -2012.224} C_VEL
LIN {X 0,Y 573.218,Z 312.703,A -85,B 0,C 180,E1 -2014.768,E2 -2014.768} C_VEL
LIN {X 0,Y 573.192,Z 312.709,A -85,B 0,C 180,E1 -2017.811,E2 -2017.811} C_VEL
LIN {X 0,Y 573.203,Z 312.703,A -85,B 0,C 180,E1 -2020.529,E2 -2020.529} C_VEL
LIN {X 0,Y 573.194,Z 312.715,A -85,B 0,C 180,E1 -2023.364,E2 -2023.364} C_VEL
LIN {X 0,Y 573.185,Z 312.706,A -85,B 0,C 180,E1 -2026.338,E2 -2026.338} C_VEL
LIN {X 0,Y 573.168,Z 312.709,A -85,B 0,C 180,E1 -2028.537,E2 -2028.537} C_VEL
LIN {X 0,Y 573.176,Z 312.717,A -85,B 0,C 180,E1 -2031.293,E2 -2031.293} C_VEL
LIN {X 0,Y 573.179,Z 312.708,A -85,B 0,C 180,E1 -2034.024,E2 -2034.024} C_VEL
LIN {X 0,Y 573.209,Z 312.705,A -85,B 0,C 180,E1 -2036.514,E2 -2036.514} C_VEL
LIN {X 0,Y 573.204,Z 312.714,A -85,B 0,C 180,E1 -2039.123,E2 -2039.123} C_VEL
LIN {X 0,Y 573.199,Z 312.707,A -85,B 0,C 180,E1 -2041.982,E2 -2041.982} C_VEL
LIN {X 0,Y 573.264,Z 312.849,A -85,B 0,C 180,E1 -2043.664,E2 -2043.664} C_VEL
LIN {X 0,Y 573.774,Z 318.807,A -85,B 0,C 180,E1 -2044.614,E2 -2044.614} C_VEL
LIN {X 0,Y 573.565,Z 337.451,A -85,B 0,C 180,E1 -2047.486,E2 -2047.486} C_VEL
LIN {X 0,Y 573.542,Z 342.75,A -85,B 0,C 180,E1 -2048.295,E2 -2048.295} C_VEL
LIN {X 0,Y 574.566,Z 348.797,A -85,B 0,C 180,E1 -2048.403,E2 -2048.403} C_VEL
LIN {X 0,Y 574.261,Z 479.98,A -85,B 0,C 180,E1 -2050.086,E2 -2050.086} C_VEL
LIN {X 0,Y 574.189,Z 494.029,A -85,B 0,C 180,E1 -2050.412,E2 -2050.412} C_VEL
LIN {X 0,Y 574.015,Z 507.978,A -85,B 0,C 180,E1 -2050.882,E2 -2050.882} C_VEL
LIN {X 0,Y 573.926,Z 520.35,A -85,B 0,C 180,E1 -2051.435,E2 -2051.435} C_VEL
LIN {X 0,Y 573.724,Z 533.314,A -85,B 0,C 180,E1 -2052.167,E2 -2052.167} C_VEL
LIN {X 0,Y 573.572,Z 545.273,A -85,B 0,C 180,E1 -2053.006,E2 -2053.006} C_VEL
LIN {X 0,Y 573.421,Z 556.773,A -85,B 0,C 180,E1 -2053.992,E2 -2053.992} C_VEL
LIN {X 0,Y 573.271,Z 567.174,A -85,B 0,C 180,E1 -2055.081,E2 -2055.081} C_VEL
LIN {X 0,Y 573.176,Z 575.74,A -85,B 0,C 180,E1 -2056.166,E2 -2056.166} C_VEL
LIN {X 0,Y 573.097,Z 583.887,A -85,B 0,C 180,E1 -2057.428,E2 -2057.428} C_VEL
LIN {X 0,Y 573.015,Z 590.414,A -85,B 0,C 180,E1 -2058.683,E2 -2058.683} C_VEL
LIN {X 0,Y 573.002,Z 594.92,A -85,B 0,C 180,E1 -2059.756,E2 -2059.756} C_VEL
LIN {X 0,Y 572.969,Z 598.445,A -85,B 0,C 180,E1 -2060.825,E2 -2060.825} C_VEL
LIN {X 0,Y 572.98,Z 601.86,A -85,B 0,C 180,E1 -2062.246,E2 -2062.246} C_VEL
LIN {X 0,Y 572.974,Z 603.858,A -85,B 0,C 180,E1 -2063.662,E2 -2063.662} C_VEL
LIN {X 0,Y 572.931,Z 604.498,A -85,B 0,C 180,E1 -2065.074,E2 -2065.074} C_VEL
LIN {X 0,Y 572.977,Z 603.796,A -85,B 0,C 180,E1 -2066.484,E2 -2066.484} C_VEL
LIN {X 0,Y 572.938,Z 601.763,A -85,B 0,C 180,E1 -2067.891,E2 -2067.891} C_VEL
LIN {X 0,Y 572.946,Z 598.349,A -85,B 0,C 180,E1 -2069.297,E2 -2069.297} C_VEL
LIN {X 0,Y 572.984,Z 593.462,A -85,B 0,C 180,E1 -2070.703,E2 -2070.703} C_VEL
LIN {X 0,Y 573.033,Z 586.957,A -85,B 0,C 180,E1 -2072.109,E2 -2072.109} C_VEL
LIN {X 0,Y 573.141,Z 579.737,A -85,B 0,C 180,E1 -2073.339,E2 -2073.339} C_VEL
LIN {X 0,Y 573.255,Z 570.831,A -85,B 0,C 180,E1 -2074.571,E2 -2074.571} C_VEL
LIN {X 0,Y 573.354,Z 561.515,A -85,B 0,C 180,E1 -2075.628,E2 -2075.628} C_VEL
LIN {X 0,Y 573.523,Z 550.066,A -85,B 0,C 180,E1 -2076.695,E2 -2076.695} C_VEL
LIN {X 0,Y 573.679,Z 538.672,A -85,B 0,C 180,E1 -2077.568,E2 -2077.568} C_VEL
LIN {X 0,Y 573.816,Z 525.911,A -85,B 0,C 180,E1 -2078.363,E2 -2078.363} C_VEL
LIN {X 0,Y 574.027,Z 512.455,A -85,B 0,C 180,E1 -2079.025,E2 -2079.025} C_VEL
LIN {X 0,Y 574.162,Z 499.548,A -85,B 0,C 180,E1 -2079.512,E2 -2079.512} C_VEL
LIN {X 0,Y 574.257,Z 485.771,A -85,B 0,C 180,E1 -2079.888,E2 -2079.888} C_VEL
LIN {X 0,Y 574.323,Z 471.488,A -85,B 0,C 180,E1 -2080.132,E2 -2080.132} C_VEL
LIN {X 0,Y 574.583,Z 348.503,A -85,B 0,C 180,E1 -2081.69,E2 -2081.69} C_VEL
LIN {X 0,Y 573.511,Z 342.677,A -85,B 0,C 180,E1 -2081.808,E2 -2081.808} C_VEL
LIN {X 0,Y 573.684,Z 324.611,A -85,B 0,C 180,E1 -2084.578,E2 -2084.578} C_VEL
LIN {X 0,Y 573.676,Z 315.467,A -85,B 0,C 180,E1 -2086,E2 -2086} C_VEL
LIN {X 0,Y 573.27,Z 312.703,A -85,B 0,C 180,E1 -2086.456,E2 -2086.456} C_VEL
LIN {X 0,Y 573.228,Z 312.707,A -85,B 0,C 180,E1 -2089.331,E2 -2089.331} C_VEL
LIN {X 0,Y 573.211,Z 312.705,A -85,B 0,C 180,E1 -2091.582,E2 -2091.582} C_VEL
LIN {X 0,Y 573.19,Z 312.706,A -85,B 0,C 180,E1 -2093.867,E2 -2093.867} C_VEL
LIN {X 0,Y 573.187,Z 312.71,A -85,B 0,C 180,E1 -2096.481,E2 -2096.481} C_VEL
LIN {X 0,Y 573.18,Z 312.712,A -85,B 0,C 180,E1 -2098.568,E2 -2098.568} C_VEL
LIN {X 0,Y 573.197,Z 312.712,A -85,B 0,C 180,E1 -2100.995,E2 -2100.995} C_VEL
LIN {X 0,Y 573.175,Z 312.708,A -85,B 0,C 180,E1 -2103.51,E2 -2103.51} C_VEL
LIN {X 0,Y 573.181,Z 312.707,A -85,B 0,C 180,E1 -2106.054,E2 -2106.054} C_VEL
LIN {X 0,Y 573.176,Z 312.717,A -85,B 0,C 180,E1 -2108.707,E2 -2108.707} C_VEL
LIN {X 0,Y 573.187,Z 312.705,A -85,B 0,C 180,E1 -2111.587,E2 -2111.587} C_VEL
LIN {X 0,Y 573.2,Z 312.709,A -85,B 0,C 180,E1 -2114.337,E2 -2114.337} C_VEL
LIN {X 0,Y 573.21,Z 312.703,A -85,B 0,C 180,E1 -2117.362,E2 -2117.362} C_VEL
LIN {X 0,Y 573.222,Z 312.711,A -85,B 0,C 180,E1 -2120.572,E2 -2120.572} C_VEL
LIN {X 0,Y 573.222,Z 312.703,A -85,B 0,C 180,E1 -2123.075,E2 -2123.075} C_VEL
LIN {X 0,Y 573.246,Z 312.698,A -85,B 0,C 180,E1 -2125.669,E2 -2125.669} C_VEL
LIN {X 0,Y 573.225,Z 312.705,A -85,B 0,C 180,E1 -2128.183,E2 -2128.183} C_VEL
LIN {X 0,Y 573.219,Z 312.708,A -85,B 0,C 180,E1 -2130.631,E2 -2130.631} C_VEL
LIN {X 0,Y 573.206,Z 312.703,A -85,B 0,C 180,E1 -2133.515,E2 -2133.515} C_VEL
LIN {X 0,Y 573.196,Z 312.71,A -85,B 0,C 180,E1 -2136.133,E2 -2136.133} C_VEL
LIN {X 0,Y 573.23,Z 312.697,A -85,B 0,C 180,E1 -2139.173,E2 -2139.173} C_VEL
LIN {X 0,Y 573.198,Z 312.703,A -85,B 0,C 180,E1 -2141.41,E2 -2141.41} C_VEL
LIN {X 0,Y 573.211,Z 312.712,A -85,B 0,C 180,E1 -2144.351,E2 -2144.351} C_VEL
LIN {X 0,Y 573.203,Z 312.708,A -85,B 0,C 180,E1 -2146.528,E2 -2146.528} C_VEL
LIN {X 0,Y 573.259,Z 312.693,A -85,B 0,C 180,E1 -2149.403,E2 -2149.403} C_VEL
LIN {X 0,Y 573.263,Z 312.705,A -85,B 0,C 180,E1 -2152.249,E2 -2152.249} C_VEL
LIN {X 0,Y 573.285,Z 312.693,A -85,B 0,C 180,E1 -2155.077,E2 -2155.077} C_VEL
LIN {X 0,Y 573.306,Z 312.697,A -85,B 0,C 180,E1 -2157.892,E2 -2157.892} C_VEL
LIN {X 0,Y 573.329,Z 312.689,A -85,B 0,C 180,E1 -2160.702,E2 -2160.702} C_VEL
LIN {X 0,Y 573.294,Z 312.693,A -85,B 0,C 180,E1 -2162.81,E2 -2162.81} C_VEL
LIN {X 0,Y 573.274,Z 312.698,A -85,B 0,C 180,E1 -2165.628,E2 -2165.628} C_VEL
LIN {X 0,Y 573.254,Z 312.7,A -85,B 0,C 180,E1 -2168.46,E2 -2168.46} C_VEL
LIN {X 0,Y 573.277,Z 312.695,A -85,B 0,C 180,E1 -2171.312,E2 -2171.312} C_VEL
LIN {X 0,Y 573.285,Z 312.696,A -85,B 0,C 180,E1 -2174.424,E2 -2174.424} C_VEL
LIN {X 0,Y 573.259,Z 312.697,A -85,B 0,C 180,E1 -2177.111,E2 -2177.111} C_VEL
LIN {X 0,Y 573.242,Z 312.705,A -85,B 0,C 180,E1 -2180.077,E2 -2180.077} C_VEL
LIN {X 0,Y 573.235,Z 312.702,A -85,B 0,C 180,E1 -2182.338,E2 -2182.338} C_VEL
LIN {X 0,Y 573.251,Z 312.702,A -85,B 0,C 180,E1 -2185.41,E2 -2185.41} C_VEL
LIN {X 0,Y 573.228,Z 312.701,A -85,B 0,C 180,E1 -2188.565,E2 -2188.565} C_VEL
LIN {X 0,Y 573.226,Z 312.702,A -85,B 0,C 180,E1 -2190.993,E2 -2190.993} C_VEL
LIN {X 0,Y 573.266,Z 312.703,A -85,B 0,C 180,E1 -2193.524,E2 -2193.524} C_VEL
LIN {X 0,Y 573.217,Z 312.706,A -85,B 0,C 180,E1 -2196.051,E2 -2196.051} C_VEL
LIN {X 0,Y 573.239,Z 312.699,A -85,B 0,C 180,E1 -2198.702,E2 -2198.702} C_VEL
LIN {X 0,Y 573.232,Z 312.71,A -85,B 0,C 180,E1 -2201.593,E2 -2201.593} C_VEL
LIN {X 0,Y 573.224,Z 312.702,A -85,B 0,C 180,E1 -2204.335,E2 -2204.335} C_VEL
LIN {X 0,Y 573.241,Z 312.707,A -85,B 0,C 180,E1 -2207.358,E2 -2207.358} C_VEL
LIN {X 0,Y 573.241,Z 312.7,A -85,B 0,C 180,E1 -2210.392,E2 -2210.392} C_VEL
LIN {X 0,Y 573.257,Z 312.702,A -85,B 0,C 180,E1 -2213.078,E2 -2213.078} C_VEL
LIN {X 0,Y 573.27,Z 312.702,A -85,B 0,C 180,E1 -2215.671,E2 -2215.671} C_VEL
LIN {X 0,Y 573.242,Z 312.7,A -85,B 0,C 180,E1 -2218.184,E2 -2218.184} C_VEL
LIN {X 0,Y 573.267,Z 312.697,A -85,B 0,C 180,E1 -2220.634,E2 -2220.634} C_VEL
LIN {X 0,Y 573.238,Z 312.709,A -85,B 0,C 180,E1 -2223.508,E2 -2223.508} C_VEL
LIN {X 0,Y 573.282,Z 312.704,A -85,B 0,C 180,E1 -2225.415,E2 -2225.415} C_VEL
LIN {X 0,Y 574.252,Z 318.098,A -85,B 0,C 180,E1 -2226.179,E2 -2226.179} C_VEL
LIN {X 0,Y 574.056,Z 336.389,A -85,B 0,C 180,E1 -2228.624,E2 -2228.624} C_VEL
LIN {X 0,Y 573.788,Z 359.12,A -85,B 0,C 180,E1 -2231.615,E2 -2231.615} C_VEL
LIN {X 0,Y 573.637,Z 371.663,A -85,B 0,C 180,E1 -2233.239,E2 -2233.239} C_VEL
LIN {X 0,Y 574.615,Z 377.462,A -85,B 0,C 180,E1 -2233.343,E2 -2233.343} C_VEL
LIN {X 0,Y 574.305,Z 508.629,A -85,B 0,C 180,E1 -2235.018,E2 -2235.018} C_VEL
LIN {X 0,Y 574.154,Z 523.393,A -85,B 0,C 180,E1 -2235.347,E2 -2235.347} C_VEL
LIN {X 0,Y 574.022,Z 537.708,A -85,B 0,C 180,E1 -2235.826,E2 -2235.826} C_VEL
LIN {X 0,Y 573.869,Z 551.642,A -85,B 0,C 180,E1 -2236.454,E2 -2236.454} C_VEL
LIN {X 0,Y 573.712,Z 564.099,A -85,B 0,C 180,E1 -2237.172,E2 -2237.172} C_VEL
LIN {X 0,Y 573.533,Z 576.642,A -85,B 0,C 180,E1 -2238.066,E2 -2238.066} C_VEL
LIN {X 0,Y 573.437,Z 588.177,A -85,B 0,C 180,E1 -2239.084,E2 -2239.084} C_VEL
LIN {X 0,Y 573.239,Z 597.851,A -85,B 0,C 180,E1 -2240.117,E2 -2240.117} C_VEL
LIN {X 0,Y 573.202,Z 606.172,A -85,B 0,C 180,E1 -2241.184,E2 -2241.184} C_VEL
LIN {X 0,Y 573.11,Z 614.127,A -85,B 0,C 180,E1 -2242.425,E2 -2242.425} C_VEL
LIN {X 0,Y 573.02,Z 620.527,A -85,B 0,C 180,E1 -2243.663,E2 -2243.663} C_VEL
LIN {X 0,Y 573.001,Z 624.961,A -85,B 0,C 180,E1 -2244.722,E2 -2244.722} C_VEL
LIN {X 0,Y 573.028,Z 628.443,A -85,B 0,C 180,E1 -2245.78,E2 -2245.78} C_VEL
LIN {X 0,Y 572.956,Z 631.832,A -85,B 0,C 180,E1 -2247.188,E2 -2247.188} C_VEL
LIN {X 0,Y 572.941,Z 633.833,A -85,B 0,C 180,E1 -2248.594,E2 -2248.594} C_VEL
LIN {X 0,Y 572.937,Z 634.5,A -85,B 0,C 180,E1 -2250,E2 -2250} C_VEL
LIN {X 0,Y 572.941,Z 633.833,A -85,B 0,C 180,E1 -2251.406,E2 -2251.406} C_VEL
LIN {X 0,Y 572.956,Z 631.833,A -85,B 0,C 180,E1 -2252.812,E2 -2252.812} C_VEL
LIN {X 0,Y 573.028,Z 628.444,A -85,B 0,C 180,E1 -2254.22,E2 -2254.22} C_VEL
LIN {X 0,Y 573.059,Z 623.568,A -85,B 0,C 180,E1 -2255.631,E2 -2255.631} C_VEL
LIN {X 0,Y 573.058,Z 618.851,A -85,B 0,C 180,E1 -2256.693,E2 -2256.693} C_VEL
LIN {X 0,Y 573.126,Z 612.037,A -85,B 0,C 180,E1 -2257.93,E2 -2257.93} C_VEL
LIN {X 0,Y 573.225,Z 603.558,A -85,B 0,C 180,E1 -2259.171,E2 -2259.171} C_VEL
LIN {X 0,Y 573.304,Z 594.706,A -85,B 0,C 180,E1 -2260.239,E2 -2260.239} C_VEL
LIN {X 0,Y 573.462,Z 583.989,A -85,B 0,C 180,E1 -2261.308,E2 -2261.308} C_VEL
LIN {X 0,Y 573.617,Z 573.14,A -85,B 0,C 180,E1 -2262.201,E2 -2262.201} C_VEL
LIN {X 0,Y 573.741,Z 561.255,A -85,B 0,C 180,E1 -2263.008,E2 -2263.008} C_VEL
LIN {X 0,Y 573.945,Z 548.092,A -85,B 0,C 180,E1 -2263.724,E2 -2263.724} C_VEL
LIN {X 0,Y 574.08,Z 534.813,A -85,B 0,C 180,E1 -2264.285,E2 -2264.285} C_VEL
LIN {X 0,Y 574.205,Z 520.743,A -85,B 0,C 180,E1 -2264.722,E2 -2264.722} C_VEL
LIN {X 0,Y 574.302,Z 507.121,A -85,B 0,C 180,E1 -2265.005,E2 -2265.005} C_VEL
LIN {X 0,Y 574.528,Z 376.502,A -85,B 0,C 180,E1 -2266.672,E2 -2266.672} C_VEL
LIN {X 0,Y 573.623,Z 371.497,A -85,B 0,C 180,E1 -2266.778,E2 -2266.778} C_VEL
LIN {X 0,Y 573.866,Z 351.074,A -85,B 0,C 180,E1 -2269.438,E2 -2269.438} C_VEL
LIN {X 0,Y 574.162,Z 329.445,A -85,B 0,C 180,E1 -2272.3,E2 -2272.3} C_VEL
LIN {X 0,Y 574.253,Z 318.093,A -85,B 0,C 180,E1 -2273.821,E2 -2273.821} C_VEL
LIN {X 0,Y 573.3,Z 312.702,A -85,B 0,C 180,E1 -2274.585,E2 -2274.585} C_VEL
LIN {X 0,Y 573.25,Z 312.705,A -85,B 0,C 180,E1 -2276.976,E2 -2276.976} C_VEL
LIN {X 0,Y 573.25,Z 312.699,A -85,B 0,C 180,E1 -2279.489,E2 -2279.489} C_VEL
LIN {X 0,Y 573.255,Z 312.707,A -85,B 0,C 180,E1 -2282.645,E2 -2282.645} C_VEL
LIN {X 0,Y 573.211,Z 312.705,A -85,B 0,C 180,E1 -2285.188,E2 -2285.188} C_VEL
LIN {X 0,Y 573.236,Z 312.701,A -85,B 0,C 180,E1 -2287.808,E2 -2287.808} C_VEL
LIN {X 0,Y 573.247,Z 312.708,A -85,B 0,C 180,E1 -2290.525,E2 -2290.525} C_VEL
LIN {X 0,Y 573.238,Z 312.699,A -85,B 0,C 180,E1 -2293.36,E2 -2293.36} C_VEL
LIN {X 0,Y 573.238,Z 312.706,A -85,B 0,C 180,E1 -2296.641,E2 -2296.641} C_VEL
LIN {X 0,Y 573.248,Z 312.698,A -85,B 0,C 180,E1 -2299.475,E2 -2299.475} C_VEL
